// TIA Portal V19 program export: 1 tag tables, 0 data types, 17 data blocks, 13 code blocks (in call order from the OBs), 101 instance data blocks

VAR_GLOBAL   // PLC tag table "Default tag table"
   EMG_STOP AT %I0.0 : Bool;
   HOOTER_RESET AT %I0.1 : Bool;
   POWER_FAIL AT %I0.2 : Bool;
   "AIR PRESSURE FAIL" AT %I0.3 : Bool;
   "CENTRIFUGAL_PUMP-1_TRIP_(FWD)" AT %I0.4 : Bool;
   "CENTRIFUGAL_PUMP-2_TRIP_(RET)" AT %I0.5 : Bool;
   "FLOW SWITCH-1" AT %I0.6 : Bool;
   "FLOW SWITCH-2" AT %I0.7 : Bool;
   "LEVEL_SWITCH-1" AT %I1.0 : Bool;
   "LEVEL_SWITCH-2" AT %I1.1 : Bool;
   "LEVEL_SWITCH-3" AT %I1.2 : Bool;
   "LEVEL_SWITCH-4" AT %I1.3 : Bool;
   SPARE_DI1 AT %I1.4 : Bool;
   SPARE_DI2 AT %I1.5 : Bool;
   "CENTRIFUGAL_PUMP-1(FWD)" AT %Q0.0 : Bool;
   "CENTRIFUGAL_PUMP-2(RET)" AT %Q0.1 : Bool;
   "DOSING_PUMP-1" AT %Q0.2 : Bool;
   SPARE_DO1 AT %Q0.3 : Bool;
   HOOTER AT %Q0.4 : Bool;
   "PBV-125 PURIFIED WATER VESSEL OUTLET VALVE" AT %Q0.5 : Bool;
   "PBV-126 SOFT WATER VESSEL OUTLET VALVE" AT %Q0.6 : Bool;
   "PBV-127 PW INLET LINE" AT %Q0.7 : Bool;
   "PBV-128 PURIFIED WATER VESSEL–SPRAY BALL INLET LINE" AT %Q1.0 : Bool;
   "PBV-129 SOFT WATER VESSEL INLET LINE" AT %Q1.1 : Bool;
   "LEVEL_SWITCH-10" AT %I8.0 : Bool;
   AIR_PRESSURE_SWITCH AT %I8.1 : Bool;
   "PNEUMATIC_VALVE-7" AT %Q8.0 : Bool;
   "PNEUMATIC_VALVE-8" AT %Q8.1 : Bool;
   "PNEUMATIC_VALVE-9" AT %Q8.2 : Bool;
   "PNEUMATIC_VALVE-10" AT %Q8.3 : Bool;
   "PNEUMATIC_VALVE-11" AT %Q8.4 : Bool;
   "PNEUMATIC_VALVE-12" AT %Q8.5 : Bool;
   "PNEUMATIC_VALVE-13" AT %Q8.6 : Bool;
   "PNEUMATIC_VALVE-14" AT %Q8.7 : Bool;
   "PNEUMATIC_VALVE-15" AT %Q12.0 : Bool;
   "PNEUMATIC_VALVE-16" AT %Q12.1 : Bool;
   "PNEUMATIC_VALVE-17" AT %Q12.2 : Bool;
   "PNEUMATIC_VALVE-18" AT %Q12.3 : Bool;
   "PNEUMATIC_VALVE-19" AT %Q12.4 : Bool;
   CT_SENSOR AT %IW128 : Int;
   TS_SENSOR_1 AT %IW130 : Int;
   TS_SENSOR_2 AT %IW132 : Int;
   "CENTRIFUGAL_PUMP-1_RPM" AT %QW128 : Int;
   "DOSING_PUMP-1(4-20mA)" AT %QW130 : Int;
   System_Byte AT %MB1 : Byte;
   FirstScan AT %M1.0 : Bool;
   DiagStatusUpdate AT %M1.1 : Bool;
   AlwaysTRUE AT %M1.2 : Bool;
   AlwaysFALSE AT %M1.3 : Bool;
   "PNEUMATIC_VALVE-20" AT %Q12.5 : Bool;
   "PNEUMATIC_VALVE-21" AT %Q12.6 : Bool;
   "PNEUMATIC_VALVE-22" AT %Q12.7 : Bool;
   "PZDV-1" AT %Q13.0 : Bool;
   "PZDV-2" AT %Q13.1 : Bool;
   "CIP IN" AT %Q13.2 : Bool;
   "CIP OUT" AT %Q13.3 : Bool;
   "PH NOT ACHIEVED POPUP" AT %M100.0 : Bool;
   "PH ACHIEVED POPUP" AT %M100.1 : Bool;
   ALARM_1 AT %M20.0 : Bool;
   P_TRIG AT %M300.0 : Bool;
   ALARM_2 AT %M20.1 : Bool;
   ALARM_3 AT %M20.2 : Bool;
   ALARM_4 AT %M20.3 : Bool;
   ALARM_5 AT %M20.4 : Bool;
   P_TRIG_1 AT %M300.1 : Bool;
   P_TRIG_2 AT %M300.2 : Bool;
   P_TRIG_3 AT %M300.3 : Bool;
   P_TRIG_4 AT %M300.4 : Bool;
   P_TRIG_5 AT %M300.5 : Bool;
   ALARM_6 AT %M20.5 : Bool;
   ALARM_7 AT %M20.6 : Bool;
   P_TRIG_6 AT %M300.6 : Bool;
   P_TRIG_7 AT %M300.7 : Bool;
   ALARM_8 AT %M20.7 : Bool;
   P_TRIG_8 AT %M301.0 : Bool;
   P_TRIG_9 AT %M301.1 : Bool;
   "RINSE-1_START_POPUP" AT %M2.0 : Bool;
   "RINSE-1 RECIRCULATION_OR_DRAIN" AT %M2.1 : Bool;
   PH_ACHIEVED AT %M2.3 : Bool;
   "RINSE-2_START_POPUP" AT %M2.5 : Bool;
   PH_NOT_ACHIEVED AT %M2.4 : Bool;
   POPUPS AT %MW2 : Word;
   "FRESH CYCLE BIT" AT %M70.0 : Bool;
   "HEATING TEMPERATURE" AT %MD4 : Real;
   "HYSTERSIS ANS" AT %MD8 : Real;
   "HEATING BIT ON" AT %M70.1 : Bool;
   Tag_1 AT %QW96 : Int;
   "PUPM-1_SPEED" AT %MD12 : Real;
   ALARM AT %MW200 : Word;
   "ALAKLI / ACID_START" AT %M2.2 : Bool;
   "RINSE-2_RECIRCULATE_OR_DRAIN" AT %M2.6 : Bool;
   "RINSE-3_RECIRCULATION_OR_DRAIN" AT %M3.0 : Bool;
   FINAL_RINSE_START AT %M3.1 : Bool;
   CONDUCTIVITY_ACHIEVED AT %M3.2 : Bool;
   CONDUCTIVITY_NOT_ACHIEVED_RECIRCULATION_OR_FRESH_CYCLE AT %M3.3 : Bool;
   GOING_TO_FRESH_CYCLE AT %M3.4 : Bool;
   ALARM_9 AT %M21.0 : Bool;
   ERROR AT %M80.0 : Bool;
   "REST TESTYT" AT %M11.0 : Bool;
   PTRIG_10 AT %M11.1 : Bool;
   "RINSE-3_START" AT %M2.7 : Bool;
   ALKALI_LOW_LEVEL_POPUP AT %M3.5 : Bool;
   ACID_LOW_LEVEL_POPUP AT %M3.6 : Bool;
   RESET AT %M0.0 : Bool;
   ALKALI_BIT AT %M0.1 : Bool;
   ACID_BIT AT %M0.2 : Bool;
   "ALAKLI / ACID FRESH CYCLE" AT %M0.3 : Bool;
   "ALKALI/ ACID SELECT_POPUP" AT %M3.7 : Bool;
   "ALKALI / ACID DRAIN_SET" AT %M0.4 : Bool;
   FINAL_RINSE_DRAIN_SET AT %M0.5 : Bool;
   CONDUCTIVITY_ACHIEVED_BIT AT %M0.6 : Bool;
   CONDUCTIVITY_NOT_ACHIEVED_BIT AT %M0.7 : Bool;
   ALARM_10 AT %M21.1 : Bool;
   CYCLE_PAUSE_LSW_FWD AT %M16.0 : Bool;
   CYCLE_PAUSE_LSW_RET AT %M16.1 : Bool;
   AUTO_RESET AT %M16.2 : Bool;
   "RINSE-1_OVER" AT %M17.0 : Bool;
   "ALKALI / ACID_OVER" AT %M17.1 : Bool;
   "RINSE-2_OVER" AT %M17.2 : Bool;
   "FINAL RINSE-1_OVER" AT %M17.3 : Bool;
   "FINAL RINSE-2_OVER" AT %M17.4 : Bool;
   PTRIG_11 AT %M16.3 : Bool;
   PTRIG_12 AT %M16.4 : Bool;
   PTRIG_13 AT %M16.5 : Bool;
   PTRIG_14 AT %M16.6 : Bool;
   PTRIG_15 AT %M16.7 : Bool;
   CYCLE_OVER_ALARM AT %MW17 : Word;
   "CYCLE PAUSE" AT %M19.0 : Bool;
   VACCUME_VALVE_AUTO_BIT AT %M19.1 : Bool;
   N_TRIG AT %M19.2 : Bool;
   P_TRIG_10 AT %M301.2 : Bool;
   ALARM_11 AT %M21.2 : Bool;
   ALARM_12 AT %M21.3 : Bool;
   P_TRIG_11 AT %M301.3 : Bool;
   PTRIG_16 AT %M19.3 : Bool;
   PTRIG_17 AT %M19.4 : Bool;
   N_TRIG1 AT %M19.5 : Bool;
   N_TRIG2 AT %M19.6 : Bool;
   "TRIGGER 1" AT %M19.7 : Bool;
   "SET PRINT BIT" AT %M21.4 : Bool;
   "TAG SET" AT %M21.5 : Bool;
   LENGTH AT %MW22 : Int;
   TRIGGER AT %M70.3 : Bool;
   "EMG TRIG" AT %M24.0 : Bool;
   "AL1 REQ" AT %M24.1 : Bool;
   "AL2 REQ" AT %M24.2 : Bool;
   POWER_TRIG AT %M24.3 : Bool;
   "AL3 REQ" AT %M24.4 : Bool;
   "FWD TRIP_TRIG" AT %M24.5 : Bool;
   "AL4 REQ" AT %M24.6 : Bool;
   "RET TRIP_TRIG" AT %M24.7 : Bool;
   "AL5 REQ" AT %M25.0 : Bool;
   ALKALI_LL_TRIG AT %M25.1 : Bool;
   "AL6 REQ" AT %M25.2 : Bool;
   ACID_LL_TRIG AT %M25.3 : Bool;
   "AL7 REQ" AT %M25.4 : Bool;
   PWT_LL_TRIG AT %M25.5 : Bool;
   "AL8 REQ" AT %M25.6 : Bool;
   SWT_LL_TRIG AT %M25.7 : Bool;
   "AL9 REQ" AT %M26.0 : Bool;
   AIR_TRIG AT %M26.1 : Bool;
   FLS_TRIG AT %M26.2 : Bool;
   "AL10 REQ" AT %M26.3 : Bool;
   "AL11 REQ" AT %M26.4 : Bool;
   RLS_TRIG AT %M26.5 : Bool;
   PRODUCT_NAME AT %IB0 : Char;
   "PROD LENGTH" AT %MW28 : Int;
   "ADD PROD LENGTH" AT %MW30 : Int;
   "EQP LENGTH" AT %MW32 : Int;
   "ADD EQP LENGTH" AT %MW34 : Int;
   "OP LENGTH" AT %MW36 : Int;
   "ADD OP LENGTH" AT %MW38 : Int;
   "BATCH LENGTH" AT %MW40 : Int;
   "BATCH ACTUAL LENGTH" AT %MW42 : Int;
   "RECIPE LENGTH" AT %MW44 : Int;
   "ADD RECIPE LENGTH" AT %MW46 : Int;
   "EMP LENGTH" AT %MW48 : Int;
   "ADD EMP LENGTH" AT %MW50 : Int;
   N_TRIG3 AT %M21.6 : Bool;
   FOOTER AT %M21.7 : Bool;
   P_TRIG20 AT %M26.6 : Bool;
   PNV25 AT %Q13.4 : Bool;
   "SW TANK_START_POPUP" AT %M27.0 : Bool;
   "PW TANK_START_POPUP" AT %M27.1 : Bool;
   "SW TANK_OVER" AT %M27.2 : Bool;
   "PW TANK_OVER" AT %M27.3 : Bool;
   P_TRIG_12 AT %M26.7 : Bool;
   P_TRIG_13 AT %M27.4 : Bool;
   xyz AT %M27.5 : Bool;
   ON AT %M27.6 : Bool;
   ON1 AT %M27.7 : Bool;
   on2 AT %M52.0 : Bool;
   on4 AT %M52.1 : Bool;
   "PASSWORD DB" AT %MW54 : Int;
   "ACK 6MONTH" AT %M52.2 : Bool;
   "ACK 8MONTH" AT %M52.3 : Bool;
   "POPUP FOR 6 MONTH" AT %M52.4 : Bool;
   "POPUP FOR 8 MONTH" AT %M52.5 : Bool;
   "POPUP BIT TRIG" AT %M52.6 : Bool;
   "PBV-130 SOFT WATER VESSEL–SPRAY BALL INLET LINE" AT %Q14.0 : Bool;
   "PBV-131 DOSING PUMP INLET LINE" AT %Q14.1 : Bool;
   "PBV-132 PURIFIED WATER VESSEL OUTLET LINE" AT %Q14.2 : Bool;
   "PBV-133 SOFT WATER VESSEL OUTLET LINE" AT %Q14.3 : Bool;
   "PBV-134 FORWARD PUMP INLET LINE" AT %Q14.4 : Bool;
   "PBV-135 REVERSE PUMP CASING DRAIN" AT %Q14.5 : Bool;
   "PBV-136 FORWARD PUMP RECIRCULATION LINE" AT %Q14.6 : Bool;
   "PBV-137 FORWARD PUMP TO HEAT EXCHANGER LINE" AT %Q14.7 : Bool;
   "PBV-138 PURIFIED WATER DRAIN LINE" AT %Q15.0 : Bool;
   "PAV-139 HEAT EXCHANGER BYPASS DRAIN" AT %Q15.1 : Bool;
   "PBV-140 HEAT EXCHANGER INLET LINE" AT %Q15.2 : Bool;
   "PAV-141 STEAM INLET LINE" AT %Q15.3 : Bool;
   "PBV-142 FORWARD PUMP RECIRCULATION LINE" AT %Q15.4 : Bool;
   "PBV-143 FORWARD PUMP TO VESSEL INLET LINE" AT %Q15.5 : Bool;
   "PBV-144 VESSEL INLET LINE" AT %Q16.0 : Bool;
   "PBV-145 REVERSE PUMP TO VESSEL RECIRCULATION LINE" AT %Q16.1 : Bool;
   "PBV-146 REVERSE PUMP TO DRAIN LINE" AT %Q16.2 : Bool;
   "PBV-147 REVERSE PUMP CASING DRAIN LINE" AT %Q16.3 : Bool;
   "PBV-148 REVERSE PUMP INLET LINE" AT %Q16.4 : Bool;
   "PBV-157 SOFT WATER DRAIN LINE" AT %Q16.5 : Bool;
   "PBV-158 SOFT WATER VENT VALVE" AT %Q16.6 : Bool;
   "PBV-159 PURIFIED VENT VALVE" AT %Q16.7 : Bool;
   "PBV-160 ALKALI VALVE" AT %Q17.0 : Bool;
   "PBV-161 ACID VALVE" AT %Q17.1 : Bool;
   SPARE_DO4 AT %Q17.2 : Bool;
   SPARE_DO5 AT %Q17.3 : Bool;
   SPARE_DO6 AT %Q17.4 : Bool;
   SPARE_DO7 AT %Q17.5 : Bool;
   SPARE_DO8 AT %Q17.6 : Bool;
   SPARE_DO9 AT %Q17.7 : Bool;
   SPARE_DO2 AT %Q15.6 : Bool;
   SPARE_DO3 AT %Q15.7 : Bool;
   PH_SENSOR AT %IW134 : Int;
END_VAR

DATA_BLOCK "BATCH DATA"   // DB171
{ S7_Optimized_Access := 'FALSE' }
   VAR
      PRODUCT_NAME : String[30] := '  PRODUCT NAME             :  ';
      PRODUCT_NAME_CONCATE : String[80];
      BATCH_NO : String[30] := '  BATCH NO                 :  ';
      BATCH_NO_CONCATE : String[80];
      EQUIPMENT_ID_NO : String[30] := '  EQUIPMENT ID NO          :  ';
      EQUIPMENT_ID_NO_CONCATE : String[80];
      RECIPE_NO : String[30] := '  RECIPE NO                :  ';
      RECIPE_NO_CONCATE : String[80];
      OPERATOR_NAME : String[30] := '  OPERATOR NAME            :  ';
      OPERATOR_NAME_CONCATE : String[80];
      EMPLOYE_CODE : String[30] := '  EMPLOYE CODE             :  ';
      EMPLOYE_CODE_CONCATE : String[80];
   END_VAR
BEGIN
END_DATA_BLOCK

DATA_BLOCK "BUFFER"   // DB26
{ S7_Optimized_Access := 'FALSE' }
   VAR
      HMI_START : Bool;
      HMI_STOP : Bool;
      "MODE SELECTION" : Int;
      PROCESS : Int;
      Static_1 : Int;
      HMI_AUTO : Bool;
      HMI_MANUAL : Bool;
      HMI_STANDBY : Bool;
      "RECIPE DOWNLOAD" : Bool;
      "LEVEL BUFFER SWT" : Int;
      "LEVEL BUFFER PWT" : Int;
      "RINSE-1" : Int;
      "ACID / ALAKLI" : Int;
      "RINSE-2" : Int;
      "RINSE-3" : Int;
      FINAL_RINSE : Int;
      CONTINUE : Bool;
      RESET : Bool;
      phMAINTAIN : Bool;
   END_VAR
BEGIN
END_DATA_BLOCK

DATA_BLOCK "CYCLE_POPUP"   // DB37
{ S7_Optimized_Access := 'FALSE' }
   VAR
      "RINSE-1_START_YES" : Bool;
      "RINSE-1_START_NO" : Bool;
      "RINSE-1_RECIRCULATION" : Bool;
      "RINSE-1_DRAIN" : Bool;
      "RINSE-2_START_YES" : Bool;
      "RINSE-2_START_NO" : Bool;
      "RINSE-2_RECIRCULATION" : Bool;
      "RINSE-2_DRAIN" : Bool;
      "ACID/ALKALI_START_YES" : Bool;
      "ACID/ALKALI_START_NO" : Bool;
      "ALKALI/ACID_RECIRCULATION" : Bool;
      "ALKALI/ACID_DRAIN" : Bool;
      "ACID/ALKALI CONTINUE CYCLE" : Bool;
      "RINSE-3_START_YES" : Bool;
      "RINSE-3_START_NO" : Bool;
      "RINSE-3_RECIRCULATION" : Bool;
      "RINSE-3_DRAIN" : Bool;
      FINAL_RINSE_START_YES : Bool;
      FINAL_RINSE_START_NO : Bool;
      FINAL_RINSE_RECIRCULATION : Bool;
      FINAL_RINSE_FRESH_CYCLE : Bool;
      ALKALI : Bool;
      ACID : Bool;
      "ALKALI /ACID FRESH CYCLE" : Bool;
      FINAL_RINSE_DRAIN : Bool;
      "SW TANK_START_YES" : Bool;
      "SW TANK_START_NO" : Bool;
      "PW TANK_START_YES" : Bool;
      "PW TANK_START_NO" : Bool;
      "PW TANK_START_YES1" : Bool;
   END_VAR
BEGIN
END_DATA_BLOCK

DATA_BLOCK "DATE& TIME_DB"   // DB10
{ S7_Optimized_Access := 'TRUE' }
// stored: MemoryReserve 100
   VAR RETAIN
      READ : DTL;
      WRITE : DTL;
   END_VAR
   VAR
      SET : Bool;
      READ_DATE : Int;
      WRITE__DATE : Int;
   END_VAR
BEGIN
END_DATA_BLOCK

DATA_BLOCK "DATE_AND_TIME"   // DB5
{ S7_Optimized_Access := 'FALSE' }
   VAR
      SET_YEAR : DWord;
      SET_MONTH : DWord;
      SET_DAY : DWord;
      SET_HOUR : DWord;
      SET_MIN : DWord;
      SET_SEC : DWord;
   END_VAR
BEGIN
END_DATA_BLOCK

DATA_BLOCK "HEADER_DATA"   // DB170
{ S7_Optimized_Access := 'TRUE' }
// stored: MemoryReserve 100
BEGIN
END_DATA_BLOCK

DATA_BLOCK "HMI"   // DB86
{ S7_Optimized_Access := 'TRUE' }
// stored: MemoryReserve 100
   VAR
      HOOTER_RESET : Bool;
      M1_SUGAR : Bool;
      M1_MFG : Bool;
      M1_STORAGE_1 : Bool;
      M1_STORAGE_2 : Bool;
      M1_MIXING : Bool;
      M2_MFG : Bool;
      M2_STORAGE_1 : Bool;
      M2_STORAGE_2 : Bool;
      M2_MIXING : Bool;
   END_VAR
BEGIN
END_DATA_BLOCK

DATA_BLOCK "IN"   // DB28
{ S7_Optimized_Access := 'FALSE' }
   VAR
      EMG_STOP : Bool;
      HOOTER_RESET : Bool;
      POWER_FAIL : Bool;
      "PUMP-1_TRIP" : Bool;
      "PUMP-2_TRIP" : Bool;
      SWT_LL : Bool;
      SWT_ML : Bool;
      SWT_HL : Bool;
      PWT_LL : Bool;
      PWT_ML : Bool;
      PWT_HL : Bool;
      ALKALI_LL : Bool;
      ALAKLI_HL : Bool;
      ACID_LL : Bool;
      ACID_HL : Bool;
      LSW_FWD_PUMP : Bool;
      LSW_RET_PUMP : Bool;
      AIR_SWITCH : Bool;
      CT_SENSOR : Int;
      PH_SENSOR : Int;
      TEMP_SENSOR : Int;
   END_VAR
BEGIN
END_DATA_BLOCK

DATA_BLOCK "MANUAL BIT"   // DB1
{ S7_Optimized_Access := 'FALSE' }
   VAR
      HOOTER : Bool;
      "PUMP-1" : Bool;
      "PUMP-2" : Bool;
      DS_PUMP : Bool;
      "PNV-1" : Bool;
      "PNV-2" : Bool;
      "PNV-3" : Bool;
      "PNV-4" : Bool;
      "PNV-5" : Bool;
      "PNV-6" : Bool;
      "PNV-7" : Bool;
      "PNV-8" : Bool;
      "PNV-9" : Bool;
      "PNV-10" : Bool;
      "PNV-11" : Bool;
      "PNV-12" : Bool;
      "PNV-13" : Bool;
      "PNV-14" : Bool;
      "PNV-15" : Bool;
      "PNV-16" : Bool;
      "PNV-17" : Bool;
      "PNV-18" : Bool;
      "PNV-19" : Bool;
      "PNV-20" : Bool;
      "PNV-21" : Bool;
      "PNV-22" : Bool;
      "PZDV-1" : Bool;
      "PZDV-2" : Bool;
      CIP_IN : Bool;
      CIP_OUT : Bool;
      "PNV-25" : Bool;
   END_VAR
BEGIN
END_DATA_BLOCK

DATA_BLOCK "MODE SELECTION"   // DB27
{ S7_Optimized_Access := 'FALSE' }
   VAR
      AUTO : Bool;
      MANUAL : Bool;
      STANDBY : Bool;
      "MODE BUFFER" : Int;
   END_VAR
BEGIN
END_DATA_BLOCK

DATA_BLOCK "OP"   // DB29
{ S7_Optimized_Access := 'FALSE' }
   VAR
      HOOTER : Bool;
      "PUMP-1" : Bool;
      "PUMP-2" : Bool;
      DS_PUMP : Bool;
      "PNV-1" : Bool;
      "PNV-2" : Bool;
      "PNV-3" : Bool;
      "PNV-4" : Bool;
      "PNV-5" : Bool;
      "PNV-6" : Bool;
      "PNV-7" : Bool;
      "PNV-8" : Bool;
      "PNV-9" : Bool;
      "PNV-10" : Bool;
      "PNV-11" : Bool;
      "PNV-12" : Bool;
      "PNV-13" : Bool;
      "PNV-14" : Bool;
      "PNV-15" : Bool;
      "PNV-16" : Bool;
      "PNV-17" : Bool;
      "PNV-18" : Bool;
      "PNV-19" : Bool;
      "PNV-20" : Bool;
      "PNV-21" : Bool;
      "PNV-22" : Bool;
      "PZDV-1" : Bool;
      "PZDV-2" : Bool;
      CIP_IN : Bool;
      CIP_OUT : Bool;
      "PNV-25" : Bool;
   END_VAR
BEGIN
END_DATA_BLOCK

DATA_BLOCK "PRINT"   // DB134
{ S7_Optimized_Access := 'TRUE' }
// stored: MemoryReserve 100
   VAR RETAIN
      "PRINT START" : Bool;
   END_VAR
   VAR
      "PRESENT VALUE" : Int;
   END_VAR
   VAR RETAIN
      INTERVAL : Int;
   END_VAR
BEGIN
END_DATA_BLOCK

DATA_BLOCK "PRINTING DATA"   // DB133
{ S7_Optimized_Access := 'FALSE' }
   VAR
      "LINE 1" : String[80] := '                          M/S PHARMAFORCE LAB UNIT-II                       ';
      "LINE 2" : String[80] := '                 MFG BY : KOTHARI PHARMA TECHNOLOGIES  PVT LTD              ';
      "LINE 3" : String[80] := ' -------------------------------------------------------------------------------';
      "LINE 4" : String[80] := '                                     CIP SKID                                 ';
      "LINE 5" : String[80] := ' -------------------------------------------------------------------------------';
      "LINE 6" : String[80] := '    /  /              RINSE-1,RINSE-2, FINAL RINSE-1 PARAMETER    ';
      "LINE 7" : String[80] := ' -------------------------------------------------------------------------------';
      "LINE 8" : String[80] := '  PARAMETER                        SET VALUE';
      "LINE 9" : String[80] := '                                   RINSE-1          RINSE-2          F_RINSE-1';
      "LINE 10" : String[80] := '  HEATING TEMPERATURE  ';
      "LINE 11" : String[80] := '  CLEANING TIME ';
      "LINE 12" : String[80] := '  RECIRCULATION TIME ';
      "LINE 13" : String[80] := '  DRAIN TIME';
      "LINE 14" : String[80] := '  PUMP CASING DRAIN TIME ';
      "LINE 15" : String[80] := '  FWD PUMP HEATING RPM ';
      "LINE 16" : String[80] := '  FWD PUMP CLEANING RPM ';
      "LINE 17" : String[80];
      "LINE 18" : String[80] := ' -------------------------------------------------------------------------------';
      "LINE 19" : String[80] := '    /  /              ALKALI / ACID PARAMETER ';
      "LINE 20" : String[80] := ' -------------------------------------------------------------------------------';
      "LINE 21" : String[80] := '  PARAMETER                             SET VALUE                 ';
      "LINE 22" : String[80] := '  HEATING TEMPERATURE  ';
      "LINE 23" : String[80] := '  CLEANING TIME ';
      "LINE 24" : String[80] := '  RECIRCULATION TIME ';
      "LINE 25" : String[80] := '  DRAIN TIME';
      "LINE 26" : String[80] := '  PUMP CASING DRAIN TIME ';
      "LINE 27" : String[80] := '  FWD PUMP HEATING RPM ';
      "LINE 28" : String[80] := '  FWD PUMP CLEANING RPM ';
      "LINE 29" : String[80] := '  BEFORE CLEANING PH LOW ';
      "LINE 30" : String[80] := '  BEFORE CLEANING PH HIGH ';
      "LINE 31" : String[80] := '  AFTER CLEANING PH LOW ';
      "LINE 32" : String[80] := '  AFTER CLEANING PH HIGH ';
      "LINE 33" : String[80];
      "LINE 34" : String[80] := ' -------------------------------------------------------------------------------';
      "LINE 35" : String[80] := '    /  /              FINAL RINSE-2 PARAMETER    ';
      "LINE 36" : String[80] := ' -------------------------------------------------------------------------------';
      "LINE 37" : String[80] := '  PARAMETER                            SET VALUE                   ';
      "LINE 38" : String[80] := '  HEATING TEMPERATURE  ';
      "LINE 39" : String[80] := '  CLEANING TIME ';
      "LINE 40" : String[80] := '  RECIRCULATION TIME ';
      "LINE 41" : String[80] := '  DRAIN TIME';
      "LINE 42" : String[80] := '  PUMP CASING DRAIN TIME ';
      "LINE 43" : String[80] := '  FWD PUMP HEATING RPM ';
      "LINE 44" : String[80] := '  FWD PUMP CLEANING RPM ';
      "LINE 45" : String[80] := '  CONDUCTIVITY ';
      "LINE 46" : String[80];
      "LINE 47" : String[80];
      AL1 : String[80] := '      :  :        EMERGENCY PRESSED ';
      AL2 : String[80] := '      :  :        POWER FAIL ';
      AL3 : String[80] := '      :  :        FORWARD PUMP TRIP';
      AL4 : String[80] := '      :  :        RETURN PUMP TRIP';
      AL5 : String[80] := '      :  :        ALKALI LEVEL IS LOW';
      AL6 : String[80] := '      :  :        ACID LEVEL IS LOW';
      AL7 : String[80] := '      :  :        PURE WATER LEVLE IS LOW ';
      AL8 : String[80] := '      :  :        SOFTWATER LEVLE IS LOW ';
      AL9 : String[80] := '      :  :        AIR FAIL';
      AL10 : String[80] := '      :  :        FORWARD LIMIT SWITCH IS UNHEALTHY';
      AL11 : String[80] := '      :  :        RETURN LIMIT SWITCH IS UNHEALTHY';
      AL12 : String[80];
      PV1 : String[80] := ' -------------------------------------------------------------------------------';
      PV2 : String[80] := '    /  /              PRESENT VALUES    ';
      PV3 : String[80] := ' -------------------------------------------------------------------------------';
      PV4 : String[80] := '                     TEMP           PUMP-1_RPM           PH          CON ';
      PV5 : String[80] := '      :  :        ';
      BLANK : String[80] := '.                                                            ';
      FOOTER1 : String[80] := '  DONE BY :                                  CHECKED BY :                  ';
   END_VAR
BEGIN
END_DATA_BLOCK

DATA_BLOCK "RECIPE DB"   // DB9
{ S7_Optimized_Access := 'FALSE' }
   VAR
      "RINSE-1_CLEANING_TIME_SV" : Int;
      "RINSE-1_RECIRCULATION_TIME_SV" : Int;
      "RINSE-1_DRAIN_TIME_SV" : Int;
      "RINSE-1_PUMP_CHASING_TIME_SV" : Int;
      "RINSE-1_TEMPERATURE_SET" : Real;
      "RINSE-1_FWD_PUMP_HEATING_RPM" : Int;
      "RINSE-1_FWD_PUMP_CLEANING_RPM" : Int;
      "RINSE-2_TEMPERATURE_SET" : Real;
      "RINSE-2_CLEANING_TIME_SV" : Int;
      "RINSE-2_RECIRCULATION_TIME_SV" : Int;
      "RINSE-2_DRAIN_TIME_SV" : Int;
      "RINSE-2_PUMP_CHASING_TIME_SV" : Int;
      "RINSE-2_FWD_PUMP_HEATING_RPM" : Int;
      "RINSE-2_FWD_PUMP_CLEANING_RPM" : Int;
      DOSING_TIME_SV : Int;
      "ALKALI/ACID_TEMPERATURE_SET" : Real;
      "ALKALI/ACID_CLEANING_TIME_SV" : Int;
      "ALKALI/ACID_RECIRCULATION_TIME_SV" : Int;
      "ALKALI/ACID_DRAIN_TIME_SV" : Int;
      "ALKALI/ACID_PUMP_CHASING_TIME_SV" : Int;
      "ALKALI/ACID_FWD_PUMP_HEATING_RPM" : Int;
      "ALKALI/ACID_FWD_PUMP_CLEANING_RPM" : Int;
      FINAL_RINSE_TEMPERATURE_SET : Real;
      FINAL_RINSE_CLEANING_TIME_SV : Int;
      FINAL_RINSE_RECIRCULATION_TIME_SV : Int;
      FINAL_RINSE_DRAIN_TIME_SV : Int;
      FINAL_RINSE_PUMP_CHASING_TIME_SV : Int;
      "FINAL_RINSE-2_FWD_PUMP_HEATING_RPM" : Int;
      "FINAL_RINSE-2_FWD_PUMP_CLEANING_RPM" : Int;
      CONDUCTIVITY_SET : Real;
      "PH_SET (NOT USED)" : Int;
      DOSING_PH_LOW : Real;
      DOSING_PH_HIGH : Real;
      "RINSE-3_TEMPERATURE_SET" : Real;
      "RINSE-3_CLEANING_TIME_SV" : Int;
      "RINSE-3_RECIRCULATION_TIME_SV" : Int;
      "RINSE-3_DRAIN_TIME_SV" : Int;
      "RINSE-3_PUMP_CHASING_TIME_SV" : Int;
      "FINAL_RINSE-1_FWD_PUMP_HEATING_RPM" : Int;
      "FINAL_RINSE-1_FWD_PUMP_CLEANING_RPM" : Int;
      SET_TEMPERATURE : Real;
      "RINSE-1_SELECT" : Bool;
      "ALKALI / ACID_SELECT" : Bool;
      "RINSE-2_SELECT" : Bool;
      "FINAL_RINSE-1_SELECT" : Bool;
      "FINAL_RINSE-2_SELECT" : Bool;
      RECIRCULATION_PH_LOW : Real;
      RECIRCULATION_PH_HIGH : Real;
      "SW TANK_SELECT" : Bool;
      "PW TANK_SELECT" : Bool;
      "SW TANK_FWD_PUMP_CLEANING_RPM" : Int;
      "PW TANK_FWD_PUMP_CLEANING_RPM" : Int;
      "SW TANK_TEMPERATURE_SET" : Real;
      "PW TANK_TEMPERATURE_SET" : Real;
      "SW TANK_CLEANING_TIME_SV" : Int;
      "SW TANK_DRAIN_TIME_SV" : Int;
      "SW TANK_PUMP_CHASING_TIME_SV" : Int;
      "PW TANK_CLEANING_TIME_SV" : Int;
      "PW TANK_DRAIN_TIME_SV" : Int;
      "PW TANK_PUMP_CHASING_TIME_SV" : Int;
   END_VAR
BEGIN
END_DATA_BLOCK

DATA_BLOCK "SCALE_SET"   // DB36
{ S7_Optimized_Access := 'FALSE' }
   VAR RETAIN
      CT_SCALE_MIN : Real;
      CT_SCALE_MAX : Real;
      PH_SCALE_MIN : Real;
      PH_SCALE_MAX : Real;
      TS_SCALE_MIN : Real;
      TS_SCALE_MAX : Real;
      CT_NORM : Real;
      PH_NORM : Real;
      TS_NORM : Real;
      CT_PV : Real;
      PH_PV : Real;
      TS_PV : Real;
      FWD_PUMP_SPEED : Real;
      HYSTERSIS : Real;
      "PUMP-1_MIN_SPEED" : Int;
      "PUMP-1_MAX_SPEED" : Int;
   END_VAR
BEGIN
END_DATA_BLOCK

DATA_BLOCK "SET_PARAMETERS"   // DB24
{ S7_Optimized_Access := 'FALSE' }
   VAR RETAIN
      "RINSE-1_CLEANING_TIME_SV" : Int;
      "RINSE-1_CLEANING_TIME_PV" : Int;
      "RINSE-1_RECIRCULATION_TIME_SV" : Int;
      "RINSE-1_RECIRCULATION_TIME_PV" : Int;
      "RINSE-1_DRAIN_TIME_SV" : Int;
      "RINSE-1_DRAIN_TIME_PV" : Int;
      "RINSE-1_PUMP_CHASING_TIME_SV" : Int;
      "RINSE-1_PUMP_CHASING_TIME_PV" : Int;
      "RINSE-1_TEMPERATURE_SET" : Real;
      "RINSE-2_TEMPERATURE_SET" : Real;
      "RINSE-2_CLEANING_TIME_SV" : Int;
      "RINSE-2_CLEANING_TIME_PV" : Int;
      "RINSE-2_RECIRCULATION_TIME_SV" : Int;
      "RINSE-2_RECIRCULATION_TIME_PV" : Int;
      "RINSE-2_DRAIN_TIME_SV" : Int;
      "RINSE-2_DRAIN_TIME_PV" : Int;
      "RINSE-2_PUMP_CHASING_TIME_SV" : Int;
      "RINSE-2_PUMP_CHASING_TIME_PV" : Int;
      DOSING_TIME_SV : Int;
      DOSING_TIME_PV : Int;
      "ALKALI/ACID_TEMPERATURE_SET" : Real;
      "ALKALI/ACID_CLEANING_TIME_SV" : Int;
      "ALKALI/ACID_CLEANING_TIME_PV" : Int;
      "ALKALI/ACID_RECIRCULATION_TIME_SV" : Int;
      "ALKALI/ACID_RECIRCULATION_TIME_PV" : Int;
      "ALKALI/ACID_DRAIN_TIME_SV" : Int;
      "ALKALI/ACID_DRAIN_TIME_PV" : Int;
      "ALKALI/ACID_PUMP_CHASING_TIME_SV" : Int;
      "ALKALI/ACID_PUMP_CHASING_TIME_PV" : Int;
      FINAL_RINSE_TEMPERATURE_SET : Real;
      FINAL_RINSE_CLEANING_TIME_SV : Int;
      FINAL_RINSE_CLEANING_TIME_PV : Int;
      FINAL_RINSE_RECIRCULATION_TIME_SV : Int;
      FINAL_RINSE_RECIRCULATION_TIME_PV : Int;
      FINAL_RINSE_DRAIN_TIME_SV : Int;
      FINAL_RINSE_DRAIN_TIME_PV : Int;
      FINAL_RINSE_PUMP_CHASING_TIME_SV : Int;
      FINAL_RINSE_PUMP_CHASING_TIME_PV : Int;
      CONDUCTIVITY_SET : Real;
      PH_SET : Real;
      DOSING_PH_LOW : Real;
      DOSING_PH_HIGH : Real;
      "RINSE-3_TEMPERATURE_SET" : Real;
      "RINSE-3_CLEANING_TIME_SV" : Int;
      "RINSE-3_CLEANING_TIME_PV" : Int;
      "RINSE-3_RECIRCULATION_TIME_SV" : Int;
      "RINSE-3_RECIRCULATION_TIME_PV" : Int;
      "RINSE-3_DRAIN_TIME_SV" : Int;
      "RINSE-3_DRAIN_TIME_PV" : Int;
      "RINSE-3_PUMP_CHASING_TIME_SV" : Int;
      "RINSE-3_PUMP_CHASING_TIME_PV" : Int;
      SET_TEMPERATURE : Real;
      "RINSE-1_FWD_PUMP_HEATING_RPM" : Int;
      "RINSE-1_FWD_PUMP_CLEANING_RPM" : Int;
      "RINSE-2_FWD_PUMP_HEATING_RPM" : Int;
      "RINSE-2_FWD_PUMP_CLEANING_RPM" : Int;
      "ALKALI/ACID_FWD_PUMP_HEATING_RPM" : Int;
      "ALKALI/ACID_FWD_PUMP_CLEANING_RPM" : Int;
      "FINAL_RINSE-2_FWD_PUMP_HEATING_RPM" : Int;
      "FINAL_RINSE-2_FWD_PUMP_CLEANING_RPM" : Int;
      "FINAL_RINSE-1_FWD_PUMP_HEATING_RPM" : Int;
      "FINAL_RINSE-1_FWD_PUMP_CLEANING_RPM" : Int;
      "PUMP-1_SPEED" : Int;
      RECIRCULATION_PH_LOW : Real;
      RECIRCULATION_PH_HIGH : Real;
      PLANT1_TANK_SELECT : Byte;
      PLANT_SELECT : Byte;
      PLANT2_TANK_SELECT : Byte;
      PLANT3_TANK_SELECT : Byte;
      "SW TANK_CLEANING_TIME_SV" : Int;
      "SW TANK_CLEANING_TIME_PV" : Int;
      "SW TANK_DRAIN_TIME_SV" : Int;
      "SW TANK_DRAIN_TIME_PV" : Int;
      "SW TANK_PUMP_CHASING_TIME_SV" : Int;
      "SW TANK_PUMP_CHASING_TIME_PV" : Int;
      "PW TANK_CLEANING_TIME_SV" : Int;
      "PW TANK_CLEANING_TIME_PV" : Int;
      "PW TANK_DRAIN_TIME_SV" : Int;
      "PW TANK_DRAIN_TIME_PV" : Int;
      "PW TANK_PUMP_CHASING_TIME_SV" : Int;
      "PW TANK_PUMP_CHASING_TIME_PV" : Int;
      "SW TANK_FWD_PUMP_CLEANING_RPM" : Int;
      "PW TANK_FWD_PUMP_CLEANING_RPM" : Int;
      "SW TANK_TEMPERATURE_SET" : Real;
      "PW TANK_TEMPERATURE_SET" : Real;
      DOSING_PH_LOW1 : Real;
      DOSING_PH_HIGH1 : Real;
   END_VAR
BEGIN
END_DATA_BLOCK

DATA_BLOCK "STRING"   // DB169
{ S7_Optimized_Access := 'FALSE' }
   VAR
      PRODUCT_NAME : String[50];
      BATCH_NO : String[50];
      EQUIPMENT_ID_NO : String[50];
      RECIPE_NO : String[50];
      OPERATOR_NAME : String[50];
      EMPLOYE_CODE : String[50];
   END_VAR
BEGIN
END_DATA_BLOCK

ORGANIZATION_BLOCK "Main"   // OB1, LAD, ProgramCycle
TITLE = "Main Program Sweep (Cycle)"
{ S7_Optimized_Access := 'TRUE' }
// stored: SetENOAutomatically false
   VAR_INPUT
      Initial_Call : Bool;   // Initial call of this OB
      Remanence : Bool;   // =True, if remanent data are available
   END_VAR
   VAR_TEMP   // added for the SCL form of the ladder/FBD networks
      _w1 : Bool;
      _w2 : Bool;
      _w3 : Bool;
      _w4 : Bool;
      _w5 : Bool;
      _w6 : Bool;
      _w7 : Bool;
      _w8 : Bool;
   END_VAR
BEGIN

REGION Network 1: MAIN BLOCK CALLING
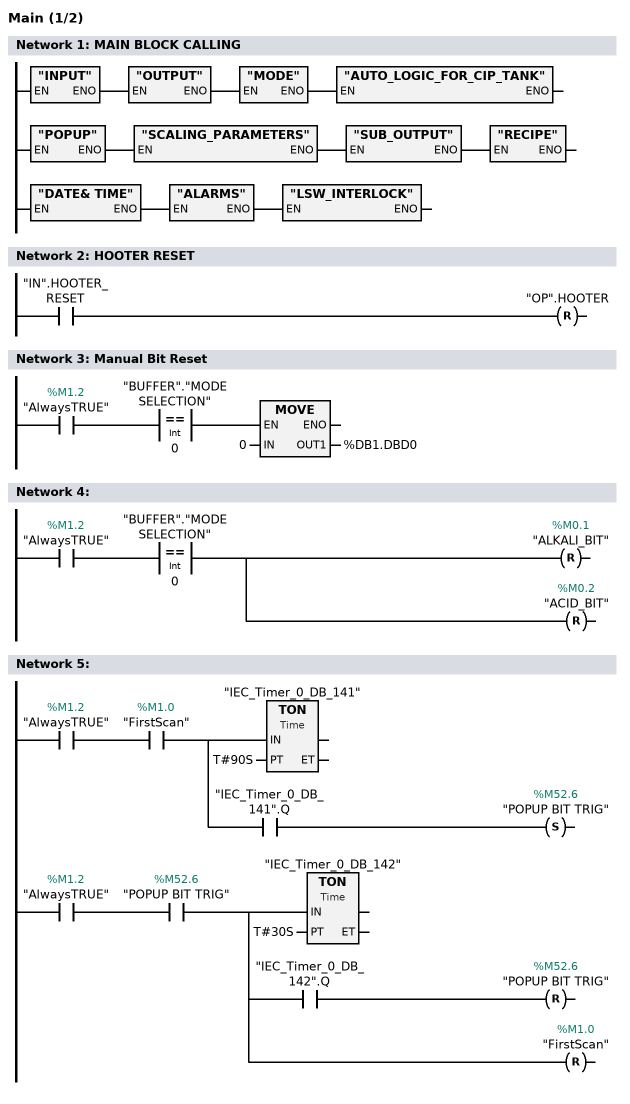
   RUNG wire#powerrail
      "INPUT"()
      "OUTPUT"()
      "MODE"()
      "AUTO_LOGIC_FOR_CIP_TANK"()
   END_RUNG
   RUNG wire#powerrail
      "POPUP"()
      "SCALING_PARAMETERS"()
      "SUB_OUTPUT"()
      "RECIPE"()
   END_RUNG
   RUNG wire#powerrail
      "DATE& TIME"()
      "ALARMS"()
      "LSW_INTERLOCK"()
   END_RUNG
   // the same network as SCL:
   "INPUT"(ENO => #_w1);
   "OUTPUT"(EN := #_w1, ENO => #_w2);
   "MODE"(EN := #_w2, ENO => #_w3);
   IF #_w3 THEN "AUTO_LOGIC_FOR_CIP_TANK"(); END_IF;
   "POPUP"(ENO => #_w4);
   "SCALING_PARAMETERS"(EN := #_w4, ENO => #_w5);
   "SUB_OUTPUT"(EN := #_w5, ENO => #_w6);
   IF #_w6 THEN "RECIPE"(); END_IF;
   "DATE& TIME"(ENO => #_w7);
   "ALARMS"(EN := #_w7, ENO => #_w8);
   IF #_w8 THEN "LSW_INTERLOCK"(); END_IF;
END_REGION

REGION Network 2: HOOTER RESET
   RUNG wire#powerrail
      Contact( "IN".HOOTER_RESET )
      R_Coil( "OP".HOOTER )
   END_RUNG
   // the same network as SCL:
   IF "IN".HOOTER_RESET THEN "OP".HOOTER := FALSE; END_IF;
END_REGION

REGION Network 3: Manual Bit Reset
   RUNG wire#powerrail
      Contact( "AlwaysTRUE" )
      { S7_Templates := "SrcType := Int" } EQ_Contact(in1 := "BUFFER"."MODE SELECTION", in2 := 0)
      Move(in := 0, out1 => %DB1.DBD0)
   END_RUNG
   // the same network as SCL:
   IF "AlwaysTRUE" AND ("BUFFER"."MODE SELECTION" = 0) THEN %DB1.DBD0 := 0; END_IF;
END_REGION

REGION Network 4
   RUNG wire#powerrail
      Contact( "AlwaysTRUE" )
      { S7_Templates := "SrcType := Int" } EQ_Contact(in1 := "BUFFER"."MODE SELECTION", in2 := 0)
      wire#w1
      R_Coil( "ALKALI_BIT" )
   END_RUNG
   RUNG wire#w1
      R_Coil( "ACID_BIT" )
   END_RUNG
   // the same network as SCL:
   IF "AlwaysTRUE" AND ("BUFFER"."MODE SELECTION" = 0) THEN
       "ALKALI_BIT" := FALSE;
       "ACID_BIT" := FALSE;
   END_IF;
END_REGION

REGION Network 5
   RUNG wire#powerrail
      Contact( "AlwaysTRUE" )
      Contact( "FirstScan" )
      wire#w1
      { S7_Templates := "time_type := Time" } "IEC_Timer_0_DB_141".TON(pt := T#90S, et =>)
   END_RUNG
   RUNG wire#w1
      Contact( "IEC_Timer_0_DB_141".Q )
      S_Coil( "POPUP BIT TRIG" )
   END_RUNG
   RUNG wire#powerrail
      Contact( "AlwaysTRUE" )
      Contact( "POPUP BIT TRIG" )
      wire#w2
      { S7_Templates := "time_type := Time" } "IEC_Timer_0_DB_142".TON(pt := T#30S, et =>)
   END_RUNG
   RUNG wire#w2
      Contact( "IEC_Timer_0_DB_142".Q )
      R_Coil( "POPUP BIT TRIG" )
   END_RUNG
   RUNG wire#w2
      R_Coil( "FirstScan" )
   END_RUNG
   // the same network as SCL:
   #_w1 := "AlwaysTRUE" AND "FirstScan";
   "IEC_Timer_0_DB_141".TON(IN := #_w1, PT := T#90S);
   IF #_w1 AND "IEC_Timer_0_DB_141".Q THEN "POPUP BIT TRIG" := TRUE; END_IF;
   #_w2 := "AlwaysTRUE" AND "POPUP BIT TRIG";
   "IEC_Timer_0_DB_142".TON(IN := #_w2, PT := T#30S);
   IF #_w2 AND "IEC_Timer_0_DB_142".Q THEN "POPUP BIT TRIG" := FALSE; END_IF;
   IF #_w2 THEN "FirstScan" := FALSE; END_IF;
END_REGION

REGION Network 6: 6 MONTH
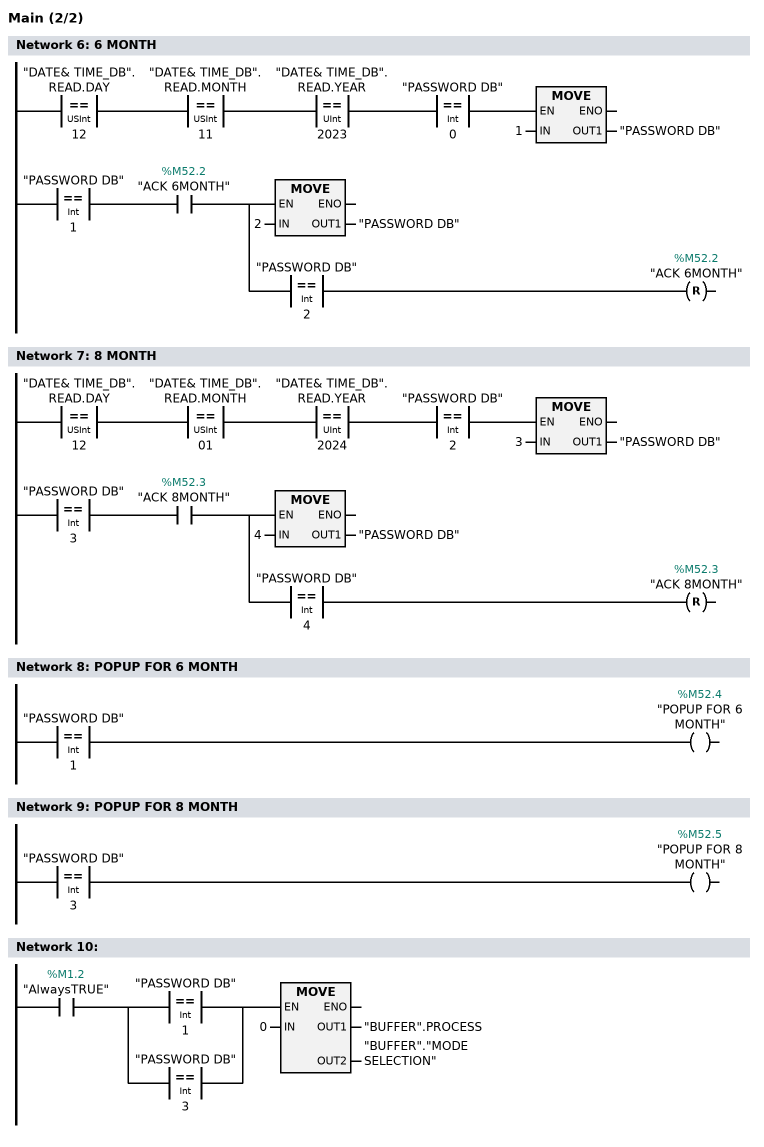
   RUNG wire#powerrail
      { S7_Templates := "SrcType := USInt" } EQ_Contact(in1 := "DATE& TIME_DB".READ.DAY, in2 := 12)
      { S7_Templates := "SrcType := USInt" } EQ_Contact(in1 := "DATE& TIME_DB".READ.MONTH, in2 := 11)
      { S7_Templates := "SrcType := UInt" } EQ_Contact(in1 := "DATE& TIME_DB".READ.YEAR, in2 := 2023)
      { S7_Templates := "SrcType := Int" } EQ_Contact(in1 := "PASSWORD DB", in2 := 0)
      Move(in := 1, out1 => "PASSWORD DB")
   END_RUNG
   RUNG wire#powerrail
      { S7_Templates := "SrcType := Int" } EQ_Contact(in1 := "PASSWORD DB", in2 := 1)
      Contact( "ACK 6MONTH" )
      wire#w1
      Move(in := 2, out1 => "PASSWORD DB")
   END_RUNG
   RUNG wire#w1
      { S7_Templates := "SrcType := Int" } EQ_Contact(in1 := "PASSWORD DB", in2 := 2)
      R_Coil( "ACK 6MONTH" )
   END_RUNG
   // the same network as SCL:
   IF ("DATE& TIME_DB".READ.DAY = 12) AND ("DATE& TIME_DB".READ.MONTH = 11) AND ("DATE& TIME_DB".READ.YEAR = 2023) AND ("PASSWORD DB" = 0) THEN
       "PASSWORD DB" := 1;
   END_IF;
   #_w1 := ("PASSWORD DB" = 1) AND "ACK 6MONTH";
   IF #_w1 THEN "PASSWORD DB" := 2; END_IF;
   IF #_w1 AND ("PASSWORD DB" = 2) THEN "ACK 6MONTH" := FALSE; END_IF;
END_REGION

REGION Network 7: 8 MONTH
   RUNG wire#powerrail
      { S7_Templates := "SrcType := USInt" } EQ_Contact(in1 := "DATE& TIME_DB".READ.DAY, in2 := 12)
      { S7_Templates := "SrcType := USInt" } EQ_Contact(in1 := "DATE& TIME_DB".READ.MONTH, in2 := 01)
      { S7_Templates := "SrcType := UInt" } EQ_Contact(in1 := "DATE& TIME_DB".READ.YEAR, in2 := 2024)
      { S7_Templates := "SrcType := Int" } EQ_Contact(in1 := "PASSWORD DB", in2 := 2)
      Move(in := 3, out1 => "PASSWORD DB")
   END_RUNG
   RUNG wire#powerrail
      { S7_Templates := "SrcType := Int" } EQ_Contact(in1 := "PASSWORD DB", in2 := 3)
      Contact( "ACK 8MONTH" )
      wire#w1
      Move(in := 4, out1 => "PASSWORD DB")
   END_RUNG
   RUNG wire#w1
      { S7_Templates := "SrcType := Int" } EQ_Contact(in1 := "PASSWORD DB", in2 := 4)
      R_Coil( "ACK 8MONTH" )
   END_RUNG
   // the same network as SCL:
   IF ("DATE& TIME_DB".READ.DAY = 12) AND ("DATE& TIME_DB".READ.MONTH = 01) AND ("DATE& TIME_DB".READ.YEAR = 2024) AND ("PASSWORD DB" = 2) THEN
       "PASSWORD DB" := 3;
   END_IF;
   #_w1 := ("PASSWORD DB" = 3) AND "ACK 8MONTH";
   IF #_w1 THEN "PASSWORD DB" := 4; END_IF;
   IF #_w1 AND ("PASSWORD DB" = 4) THEN "ACK 8MONTH" := FALSE; END_IF;
END_REGION

REGION Network 8: POPUP FOR 6 MONTH
   RUNG wire#powerrail
      { S7_Templates := "SrcType := Int" } EQ_Contact(in1 := "PASSWORD DB", in2 := 1)
      Coil( "POPUP FOR 6 MONTH" )
   END_RUNG
   // the same network as SCL:
   "POPUP FOR 6 MONTH" := "PASSWORD DB" = 1;
END_REGION

REGION Network 9: POPUP FOR 8 MONTH
   RUNG wire#powerrail
      { S7_Templates := "SrcType := Int" } EQ_Contact(in1 := "PASSWORD DB", in2 := 3)
      Coil( "POPUP FOR 8 MONTH" )
   END_RUNG
   // the same network as SCL:
   "POPUP FOR 8 MONTH" := "PASSWORD DB" = 3;
END_REGION

REGION Network 10
   RUNG wire#powerrail
      Contact( "AlwaysTRUE" )
      wire#w1
      { S7_Templates := "SrcType := Int" } EQ_Contact(in1 := "PASSWORD DB", in2 := 1)
      wire#w2
      Move(in := 0, out1 => "BUFFER".PROCESS, out2 => "BUFFER"."MODE SELECTION")
   END_RUNG
   RUNG wire#w1
      { S7_Templates := "SrcType := Int" } EQ_Contact(in1 := "PASSWORD DB", in2 := 3)
   END_RUNG wire#w2
   // the same network as SCL:
   IF "AlwaysTRUE" AND (("PASSWORD DB" = 1) OR ("PASSWORD DB" = 3)) THEN
       "BUFFER".PROCESS := 0;
       "BUFFER"."MODE SELECTION" := 0;
   END_IF;
END_REGION
END_ORGANIZATION_BLOCK

FUNCTION "INPUT" : Void   // FC2, LAD
{ S7_Optimized_Access := 'TRUE' }
// stored: SetENOAutomatically false
BEGIN

REGION Network 1: EMERGENCY_STOP
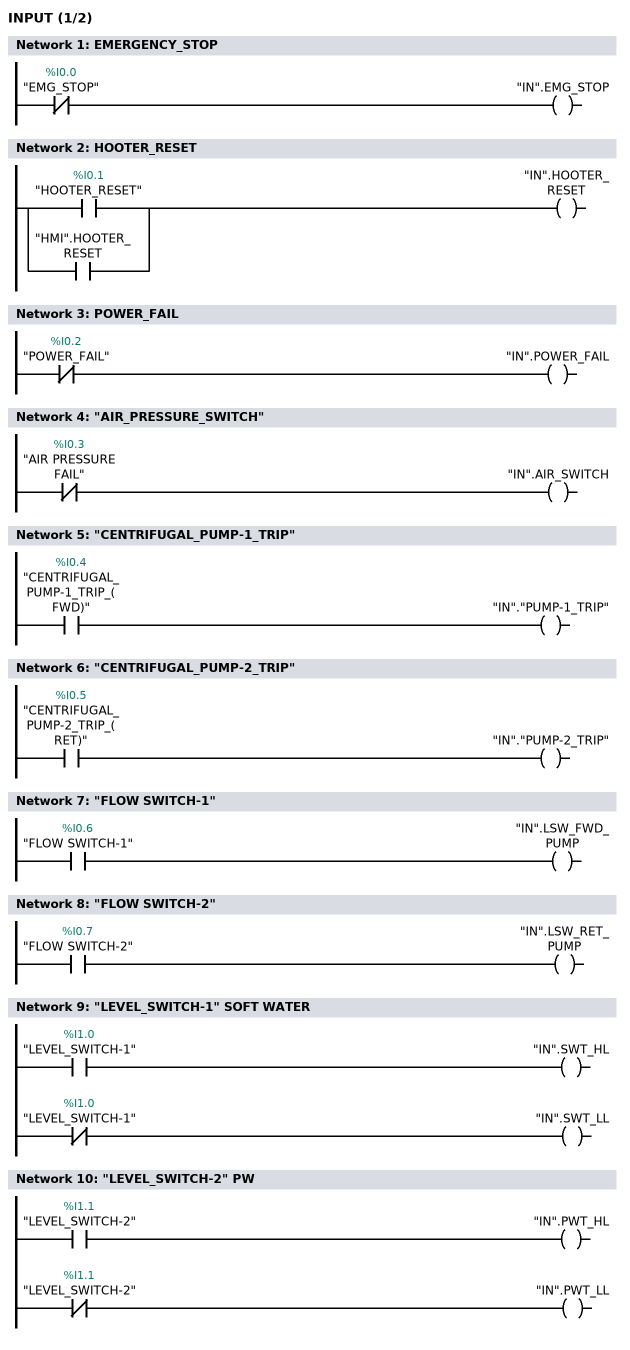
   RUNG wire#powerrail
      I_Contact( "EMG_STOP" )
      Coil( "IN".EMG_STOP )
   END_RUNG
   // the same network as SCL:
   "IN".EMG_STOP := NOT "EMG_STOP";
END_REGION

REGION Network 2: HOOTER_RESET
   RUNG wire#powerrail
      Contact( "HOOTER_RESET" )
      wire#w1
      Coil( "IN".HOOTER_RESET )
   END_RUNG
   RUNG wire#powerrail
      Contact( "HMI".HOOTER_RESET )
   END_RUNG wire#w1
   // the same network as SCL:
   "IN".HOOTER_RESET := "HOOTER_RESET" OR "HMI".HOOTER_RESET;
END_REGION

REGION Network 3: POWER_FAIL
   RUNG wire#powerrail
      I_Contact( "POWER_FAIL" )
      Coil( "IN".POWER_FAIL )
   END_RUNG
   // the same network as SCL:
   "IN".POWER_FAIL := NOT "POWER_FAIL";
END_REGION

REGION Network 4: "AIR_PRESSURE_SWITCH"
   RUNG wire#powerrail
      I_Contact( "AIR PRESSURE FAIL" )
      Coil( "IN".AIR_SWITCH )
   END_RUNG
   // the same network as SCL:
   "IN".AIR_SWITCH := NOT "AIR PRESSURE FAIL";
END_REGION

REGION Network 5: "CENTRIFUGAL_PUMP-1_TRIP"
   RUNG wire#powerrail
      Contact( "CENTRIFUGAL_PUMP-1_TRIP_(FWD)" )
      Coil( "IN"."PUMP-1_TRIP" )
   END_RUNG
   // the same network as SCL:
   "IN"."PUMP-1_TRIP" := "CENTRIFUGAL_PUMP-1_TRIP_(FWD)";
END_REGION

REGION Network 6: "CENTRIFUGAL_PUMP-2_TRIP"
   RUNG wire#powerrail
      Contact( "CENTRIFUGAL_PUMP-2_TRIP_(RET)" )
      Coil( "IN"."PUMP-2_TRIP" )
   END_RUNG
   // the same network as SCL:
   "IN"."PUMP-2_TRIP" := "CENTRIFUGAL_PUMP-2_TRIP_(RET)";
END_REGION

REGION Network 7: "FLOW SWITCH-1"
   RUNG wire#powerrail
      Contact( "FLOW SWITCH-1" )
      Coil( "IN".LSW_FWD_PUMP )
   END_RUNG
   // the same network as SCL:
   "IN".LSW_FWD_PUMP := "FLOW SWITCH-1";
END_REGION

REGION Network 8: "FLOW SWITCH-2"
   RUNG wire#powerrail
      Contact( "FLOW SWITCH-2" )
      Coil( "IN".LSW_RET_PUMP )
   END_RUNG
   // the same network as SCL:
   "IN".LSW_RET_PUMP := "FLOW SWITCH-2";
END_REGION

REGION Network 9: "LEVEL_SWITCH-1" SOFT WATER
   RUNG wire#powerrail
      Contact( "LEVEL_SWITCH-1" )
      Coil( "IN".SWT_HL )
   END_RUNG
   RUNG wire#powerrail
      I_Contact( "LEVEL_SWITCH-1" )
      Coil( "IN".SWT_LL )
   END_RUNG
   // the same network as SCL:
   "IN".SWT_HL := "LEVEL_SWITCH-1";
   "IN".SWT_LL := NOT "LEVEL_SWITCH-1";
END_REGION

REGION Network 10: "LEVEL_SWITCH-2" PW
   RUNG wire#powerrail
      Contact( "LEVEL_SWITCH-2" )
      Coil( "IN".PWT_HL )
   END_RUNG
   RUNG wire#powerrail
      I_Contact( "LEVEL_SWITCH-2" )
      Coil( "IN".PWT_LL )
   END_RUNG
   // the same network as SCL:
   "IN".PWT_HL := "LEVEL_SWITCH-2";
   "IN".PWT_LL := NOT "LEVEL_SWITCH-2";
END_REGION

REGION Network 11: "LEVEL_SWITCH-3" ALKALI
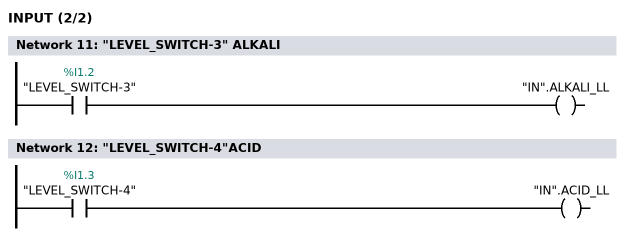
   RUNG wire#powerrail
      Contact( "LEVEL_SWITCH-3" )
      Coil( "IN".ALKALI_LL )
   END_RUNG
   // the same network as SCL:
   "IN".ALKALI_LL := "LEVEL_SWITCH-3";
END_REGION

REGION Network 12: "LEVEL_SWITCH-4"ACID
   RUNG wire#powerrail
      Contact( "LEVEL_SWITCH-4" )
      Coil( "IN".ACID_LL )
   END_RUNG
   // the same network as SCL:
   "IN".ACID_LL := "LEVEL_SWITCH-4";
END_REGION
END_FUNCTION

FUNCTION "MODE" : Void   // FC3, LAD
{ S7_Optimized_Access := 'TRUE' }
// stored: SetENOAutomatically false
   VAR_TEMP   // added for the SCL form of the ladder/FBD networks
      _w1 : Bool;
   END_VAR
BEGIN

REGION Network 1: MANUAL_MODE_SELECTION
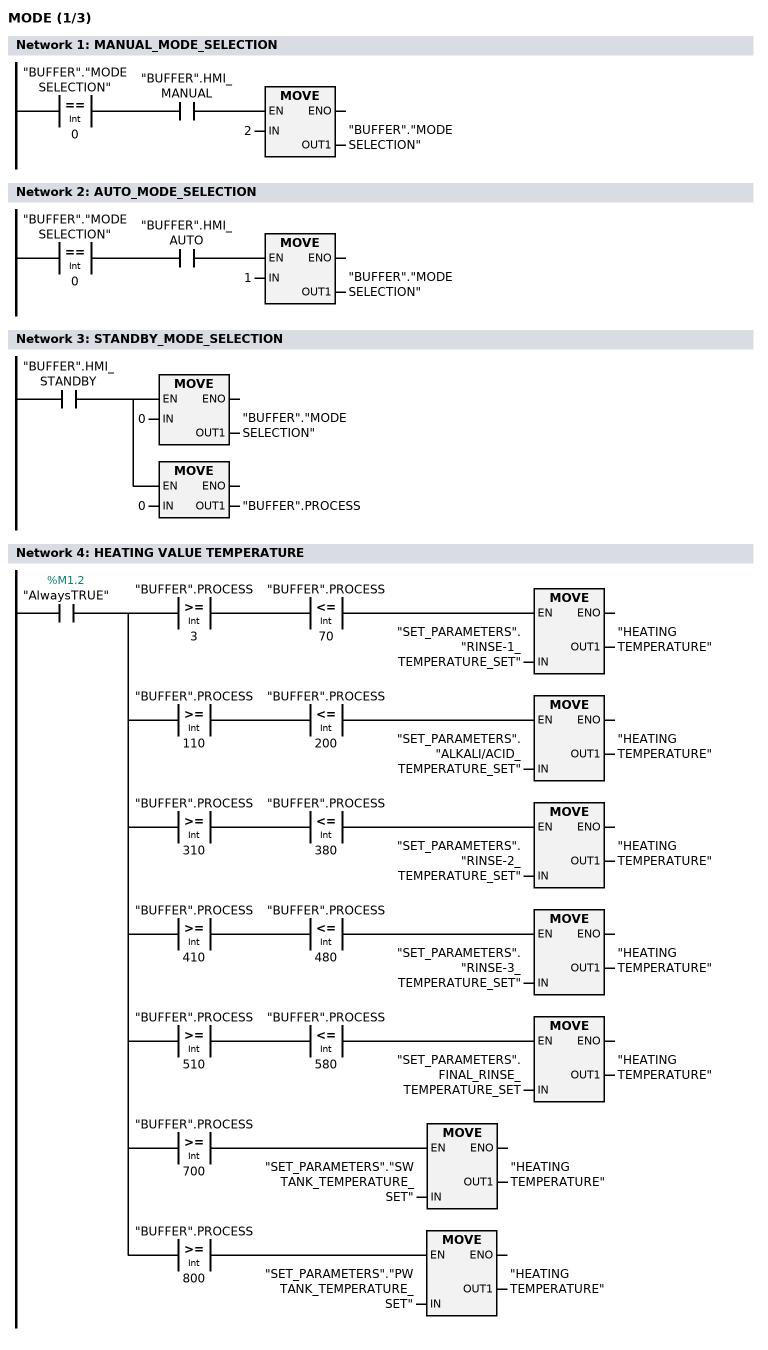
   RUNG wire#powerrail
      { S7_Templates := "SrcType := Int" } EQ_Contact(in1 := "BUFFER"."MODE SELECTION", in2 := 0)
      Contact( "BUFFER".HMI_MANUAL )
      Move(in := 2, out1 => "BUFFER"."MODE SELECTION")
   END_RUNG
   // the same network as SCL:
   IF ("BUFFER"."MODE SELECTION" = 0) AND "BUFFER".HMI_MANUAL THEN "BUFFER"."MODE SELECTION" := 2; END_IF;
END_REGION

REGION Network 2: AUTO_MODE_SELECTION
   RUNG wire#powerrail
      { S7_Templates := "SrcType := Int" } EQ_Contact(in1 := "BUFFER"."MODE SELECTION", in2 := 0)
      Contact( "BUFFER".HMI_AUTO )
      Move(in := 1, out1 => "BUFFER"."MODE SELECTION")
   END_RUNG
   // the same network as SCL:
   IF ("BUFFER"."MODE SELECTION" = 0) AND "BUFFER".HMI_AUTO THEN "BUFFER"."MODE SELECTION" := 1; END_IF;
END_REGION

REGION Network 3: STANDBY_MODE_SELECTION
   RUNG wire#powerrail
      Contact( "BUFFER".HMI_STANDBY )
      wire#w1
      Move(in := 0, out1 => "BUFFER"."MODE SELECTION")
   END_RUNG
   RUNG wire#w1
      Move(in := 0, out1 => "BUFFER".PROCESS)
   END_RUNG
   // the same network as SCL:
   IF "BUFFER".HMI_STANDBY THEN
       "BUFFER"."MODE SELECTION" := 0;
       "BUFFER".PROCESS := 0;
   END_IF;
END_REGION

REGION Network 4: HEATING VALUE TEMPERATURE
   RUNG wire#powerrail
      Contact( "AlwaysTRUE" )
      wire#w1
      { S7_Templates := "SrcType := Int" } GE_Contact(in1 := "BUFFER".PROCESS, in2 := 3)
      { S7_Templates := "SrcType := Int" } LE_Contact(in1 := "BUFFER".PROCESS, in2 := 70)
      Move(in := "SET_PARAMETERS"."RINSE-1_TEMPERATURE_SET", out1 => "HEATING TEMPERATURE")
   END_RUNG
   RUNG wire#w1
      { S7_Templates := "SrcType := Int" } GE_Contact(in1 := "BUFFER".PROCESS, in2 := 110)
      { S7_Templates := "SrcType := Int" } LE_Contact(in1 := "BUFFER".PROCESS, in2 := 200)
      Move(in := "SET_PARAMETERS"."ALKALI/ACID_TEMPERATURE_SET", out1 => "HEATING TEMPERATURE")
   END_RUNG
   RUNG wire#w1
      { S7_Templates := "SrcType := Int" } GE_Contact(in1 := "BUFFER".PROCESS, in2 := 310)
      { S7_Templates := "SrcType := Int" } LE_Contact(in1 := "BUFFER".PROCESS, in2 := 380)
      Move(in := "SET_PARAMETERS"."RINSE-2_TEMPERATURE_SET", out1 => "HEATING TEMPERATURE")
   END_RUNG
   RUNG wire#w1
      { S7_Templates := "SrcType := Int" } GE_Contact(in1 := "BUFFER".PROCESS, in2 := 410)
      { S7_Templates := "SrcType := Int" } LE_Contact(in1 := "BUFFER".PROCESS, in2 := 480)
      Move(in := "SET_PARAMETERS"."RINSE-3_TEMPERATURE_SET", out1 => "HEATING TEMPERATURE")
   END_RUNG
   RUNG wire#w1
      { S7_Templates := "SrcType := Int" } GE_Contact(in1 := "BUFFER".PROCESS, in2 := 510)
      { S7_Templates := "SrcType := Int" } LE_Contact(in1 := "BUFFER".PROCESS, in2 := 580)
      Move(in := "SET_PARAMETERS".FINAL_RINSE_TEMPERATURE_SET, out1 => "HEATING TEMPERATURE")
   END_RUNG
   RUNG wire#w1
      { S7_Templates := "SrcType := Int" } GE_Contact(in1 := "BUFFER".PROCESS, in2 := 700)
      Move(in := "SET_PARAMETERS"."SW TANK_TEMPERATURE_SET", out1 => "HEATING TEMPERATURE")
   END_RUNG
   RUNG wire#w1
      { S7_Templates := "SrcType := Int" } GE_Contact(in1 := "BUFFER".PROCESS, in2 := 800)
      Move(in := "SET_PARAMETERS"."PW TANK_TEMPERATURE_SET", out1 => "HEATING TEMPERATURE")
   END_RUNG
   // the same network as SCL:
   IF "AlwaysTRUE" AND ("BUFFER".PROCESS >= 3) AND ("BUFFER".PROCESS <= 70) THEN
       "HEATING TEMPERATURE" := "SET_PARAMETERS"."RINSE-1_TEMPERATURE_SET";
   END_IF;
   IF "AlwaysTRUE" AND ("BUFFER".PROCESS >= 110) AND ("BUFFER".PROCESS <= 200) THEN
       "HEATING TEMPERATURE" := "SET_PARAMETERS"."ALKALI/ACID_TEMPERATURE_SET";
   END_IF;
   IF "AlwaysTRUE" AND ("BUFFER".PROCESS >= 310) AND ("BUFFER".PROCESS <= 380) THEN
       "HEATING TEMPERATURE" := "SET_PARAMETERS"."RINSE-2_TEMPERATURE_SET";
   END_IF;
   IF "AlwaysTRUE" AND ("BUFFER".PROCESS >= 410) AND ("BUFFER".PROCESS <= 480) THEN
       "HEATING TEMPERATURE" := "SET_PARAMETERS"."RINSE-3_TEMPERATURE_SET";
   END_IF;
   IF "AlwaysTRUE" AND ("BUFFER".PROCESS >= 510) AND ("BUFFER".PROCESS <= 580) THEN
       "HEATING TEMPERATURE" := "SET_PARAMETERS".FINAL_RINSE_TEMPERATURE_SET;
   END_IF;
   IF "AlwaysTRUE" AND ("BUFFER".PROCESS >= 700) THEN
       "HEATING TEMPERATURE" := "SET_PARAMETERS"."SW TANK_TEMPERATURE_SET";
   END_IF;
   IF "AlwaysTRUE" AND ("BUFFER".PROCESS >= 800) THEN
       "HEATING TEMPERATURE" := "SET_PARAMETERS"."PW TANK_TEMPERATURE_SET";
   END_IF;
END_REGION

REGION Network 5: HEATING HYSTERSIS
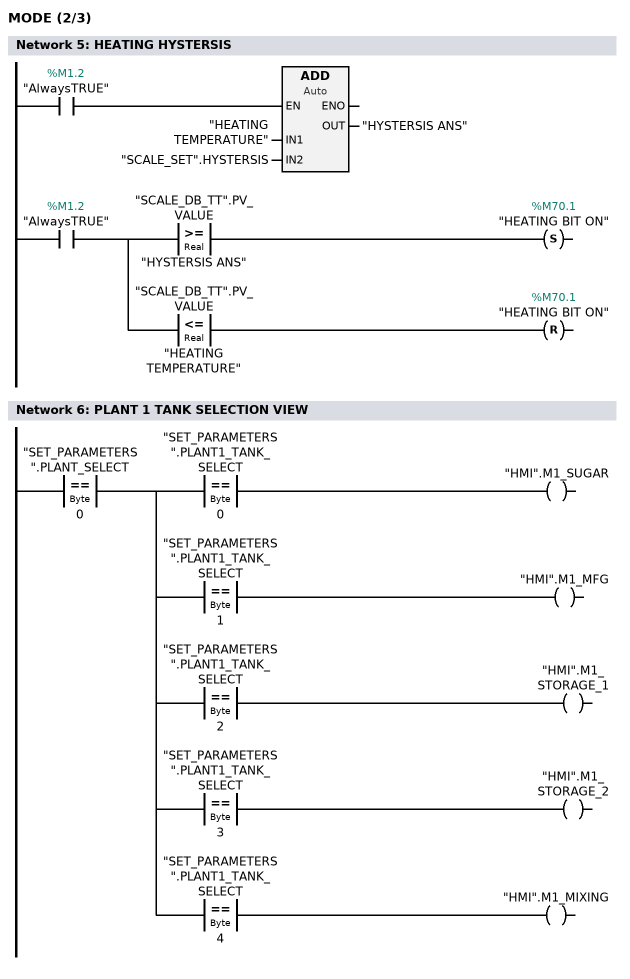
   RUNG wire#powerrail
      Contact( "AlwaysTRUE" )
      Add(in1 := "HEATING TEMPERATURE", in2 := "SCALE_SET".HYSTERSIS, out => "HYSTERSIS ANS")
   END_RUNG
   RUNG wire#powerrail
      Contact( "AlwaysTRUE" )
      wire#w1
      { S7_Templates := "SrcType := Real" } GE_Contact(in1 := "SCALE_DB_TT".PV_VALUE, in2 := "HYSTERSIS ANS")
      S_Coil( "HEATING BIT ON" )
   END_RUNG
   RUNG wire#w1
      { S7_Templates := "SrcType := Real" } LE_Contact(in1 := "SCALE_DB_TT".PV_VALUE, in2 := "HEATING TEMPERATURE")
      R_Coil( "HEATING BIT ON" )
   END_RUNG
   // the same network as SCL:
   IF "AlwaysTRUE" THEN "HYSTERSIS ANS" := "HEATING TEMPERATURE" + "SCALE_SET".HYSTERSIS; END_IF;
   IF "AlwaysTRUE" AND ("SCALE_DB_TT".PV_VALUE >= "HYSTERSIS ANS") THEN "HEATING BIT ON" := TRUE; END_IF;
   IF "AlwaysTRUE" AND ("SCALE_DB_TT".PV_VALUE <= "HEATING TEMPERATURE") THEN
       "HEATING BIT ON" := FALSE;
   END_IF;
END_REGION

REGION Network 6: PLANT 1 TANK SELECTION VIEW
   RUNG wire#powerrail
      { S7_Templates := "SrcType := Byte" } EQ_Contact(in1 := "SET_PARAMETERS".PLANT_SELECT, in2 := 0)
      wire#w1
      { S7_Templates := "SrcType := Byte" } EQ_Contact(in1 := "SET_PARAMETERS".PLANT1_TANK_SELECT, in2 := 0)
      Coil( "HMI".M1_SUGAR )
   END_RUNG
   RUNG wire#w1
      { S7_Templates := "SrcType := Byte" } EQ_Contact(in1 := "SET_PARAMETERS".PLANT1_TANK_SELECT, in2 := 1)
      Coil( "HMI".M1_MFG )
   END_RUNG
   RUNG wire#w1
      { S7_Templates := "SrcType := Byte" } EQ_Contact(in1 := "SET_PARAMETERS".PLANT1_TANK_SELECT, in2 := 2)
      Coil( "HMI".M1_STORAGE_1 )
   END_RUNG
   RUNG wire#w1
      { S7_Templates := "SrcType := Byte" } EQ_Contact(in1 := "SET_PARAMETERS".PLANT1_TANK_SELECT, in2 := 3)
      Coil( "HMI".M1_STORAGE_2 )
   END_RUNG
   RUNG wire#w1
      { S7_Templates := "SrcType := Byte" } EQ_Contact(in1 := "SET_PARAMETERS".PLANT1_TANK_SELECT, in2 := 4)
      Coil( "HMI".M1_MIXING )
   END_RUNG
   // the same network as SCL:
   #_w1 := "SET_PARAMETERS".PLANT_SELECT = 0;
   "HMI".M1_SUGAR := #_w1 AND ("SET_PARAMETERS".PLANT1_TANK_SELECT = 0);
   "HMI".M1_MFG := #_w1 AND ("SET_PARAMETERS".PLANT1_TANK_SELECT = 1);
   "HMI".M1_STORAGE_1 := #_w1 AND ("SET_PARAMETERS".PLANT1_TANK_SELECT = 2);
   "HMI".M1_STORAGE_2 := #_w1 AND ("SET_PARAMETERS".PLANT1_TANK_SELECT = 3);
   "HMI".M1_MIXING := #_w1 AND ("SET_PARAMETERS".PLANT1_TANK_SELECT = 4);
END_REGION

REGION Network 7: PLANT 2 TANK SELECTION VIEW
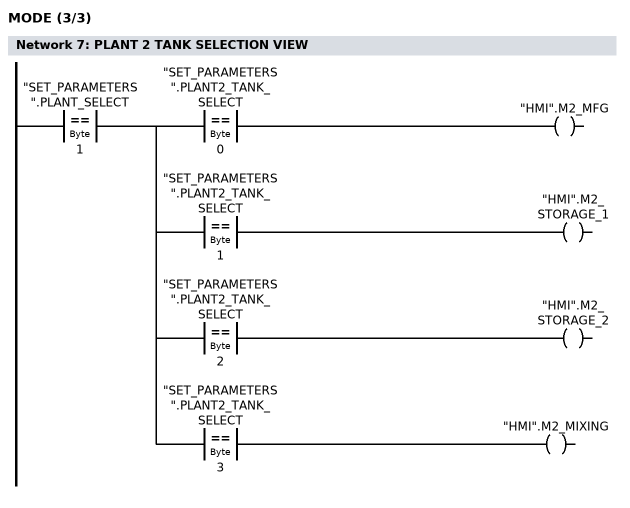
   RUNG wire#powerrail
      { S7_Templates := "SrcType := Byte" } EQ_Contact(in1 := "SET_PARAMETERS".PLANT_SELECT, in2 := 1)
      wire#w1
      { S7_Templates := "SrcType := Byte" } EQ_Contact(in1 := "SET_PARAMETERS".PLANT2_TANK_SELECT, in2 := 0)
      Coil( "HMI".M2_MFG )
   END_RUNG
   RUNG wire#w1
      { S7_Templates := "SrcType := Byte" } EQ_Contact(in1 := "SET_PARAMETERS".PLANT2_TANK_SELECT, in2 := 1)
      Coil( "HMI".M2_STORAGE_1 )
   END_RUNG
   RUNG wire#w1
      { S7_Templates := "SrcType := Byte" } EQ_Contact(in1 := "SET_PARAMETERS".PLANT2_TANK_SELECT, in2 := 2)
      Coil( "HMI".M2_STORAGE_2 )
   END_RUNG
   RUNG wire#w1
      { S7_Templates := "SrcType := Byte" } EQ_Contact(in1 := "SET_PARAMETERS".PLANT2_TANK_SELECT, in2 := 3)
      Coil( "HMI".M2_MIXING )
   END_RUNG
   // the same network as SCL:
   #_w1 := "SET_PARAMETERS".PLANT_SELECT = 1;
   "HMI".M2_MFG := #_w1 AND ("SET_PARAMETERS".PLANT2_TANK_SELECT = 0);
   "HMI".M2_STORAGE_1 := #_w1 AND ("SET_PARAMETERS".PLANT2_TANK_SELECT = 1);
   "HMI".M2_STORAGE_2 := #_w1 AND ("SET_PARAMETERS".PLANT2_TANK_SELECT = 2);
   "HMI".M2_MIXING := #_w1 AND ("SET_PARAMETERS".PLANT2_TANK_SELECT = 3);
END_REGION
END_FUNCTION

FUNCTION "AUTO_LOGIC_FOR_CIP_TANK" : Void   // FC13, LAD
{ S7_Optimized_Access := 'TRUE' }
// stored: SetENOAutomatically false
   VAR_TEMP   // added for the SCL form of the ladder/FBD networks
      _w1 : Bool;
      _w2 : Bool;
      _w3 : Bool;
      _w4 : Bool;
   END_VAR
BEGIN

REGION Network 1: START
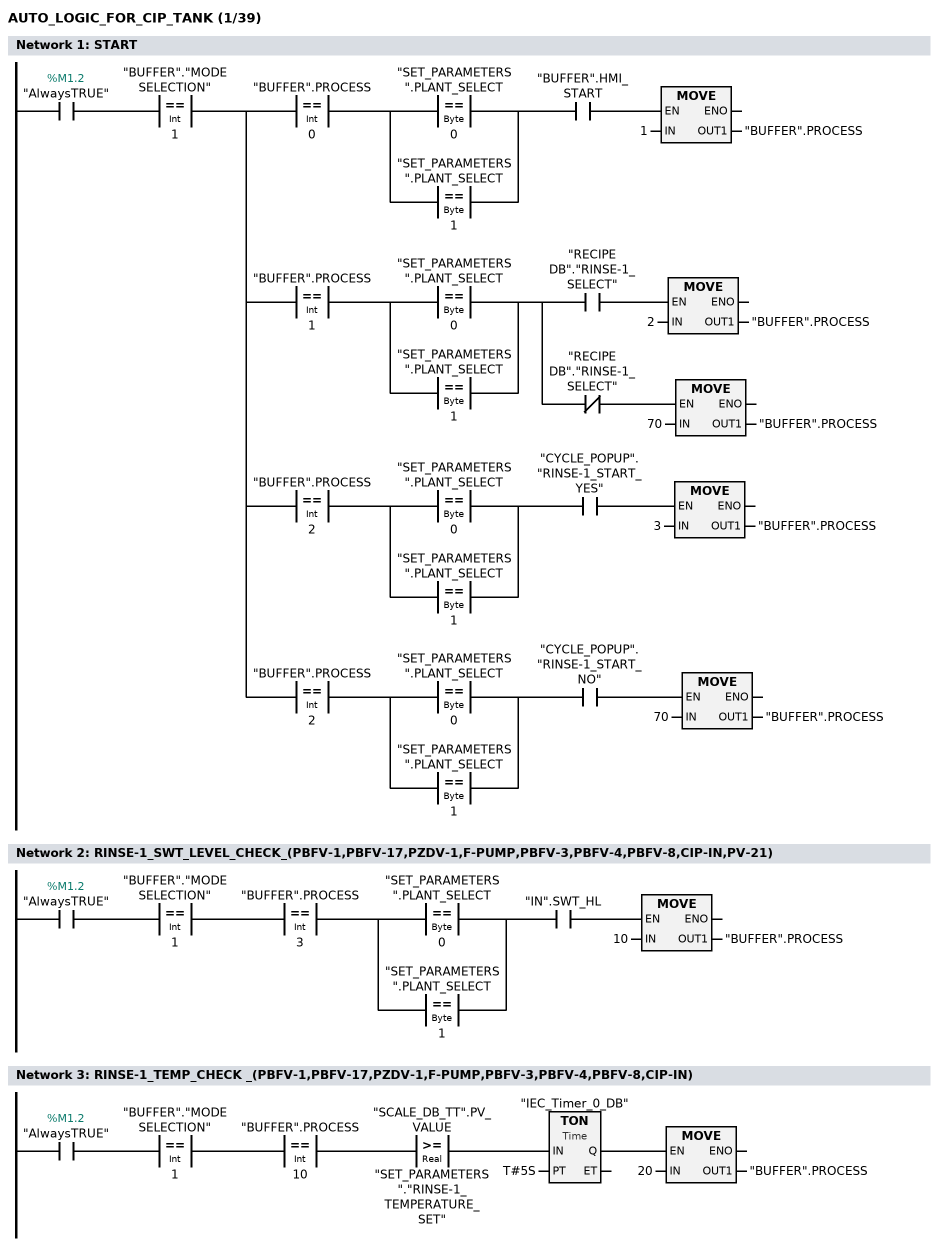
   RUNG wire#powerrail
      Contact( "AlwaysTRUE" )
      { S7_Templates := "SrcType := Int" } EQ_Contact(in1 := "BUFFER"."MODE SELECTION", in2 := 1)
      wire#w1
      { S7_Templates := "SrcType := Int" } EQ_Contact(in1 := "BUFFER".PROCESS, in2 := 0)
      wire#w2
      { S7_Templates := "SrcType := Byte" } EQ_Contact(in1 := "SET_PARAMETERS".PLANT_SELECT, in2 := 0)
      wire#w3
      Contact( "BUFFER".HMI_START )
      Move(in := 1, out1 => "BUFFER".PROCESS)
   END_RUNG
   RUNG wire#w2
      { S7_Templates := "SrcType := Byte" } EQ_Contact(in1 := "SET_PARAMETERS".PLANT_SELECT, in2 := 1)
   END_RUNG wire#w3
   RUNG wire#w1
      { S7_Templates := "SrcType := Int" } EQ_Contact(in1 := "BUFFER".PROCESS, in2 := 1)
      wire#w4
      { S7_Templates := "SrcType := Byte" } EQ_Contact(in1 := "SET_PARAMETERS".PLANT_SELECT, in2 := 0)
      wire#w5
      Contact( "RECIPE DB"."RINSE-1_SELECT" )
      Move(in := 2, out1 => "BUFFER".PROCESS)
   END_RUNG
   RUNG wire#w4
      { S7_Templates := "SrcType := Byte" } EQ_Contact(in1 := "SET_PARAMETERS".PLANT_SELECT, in2 := 1)
   END_RUNG wire#w5
   RUNG wire#w5
      I_Contact( "RECIPE DB"."RINSE-1_SELECT" )
      Move(in := 70, out1 => "BUFFER".PROCESS)
   END_RUNG
   RUNG wire#w1
      { S7_Templates := "SrcType := Int" } EQ_Contact(in1 := "BUFFER".PROCESS, in2 := 2)
      wire#w6
      { S7_Templates := "SrcType := Byte" } EQ_Contact(in1 := "SET_PARAMETERS".PLANT_SELECT, in2 := 0)
      wire#w7
      Contact( "CYCLE_POPUP"."RINSE-1_START_YES" )
      Move(in := 3, out1 => "BUFFER".PROCESS)
   END_RUNG
   RUNG wire#w6
      { S7_Templates := "SrcType := Byte" } EQ_Contact(in1 := "SET_PARAMETERS".PLANT_SELECT, in2 := 1)
   END_RUNG wire#w7
   RUNG wire#w1
      { S7_Templates := "SrcType := Int" } EQ_Contact(in1 := "BUFFER".PROCESS, in2 := 2)
      wire#w8
      { S7_Templates := "SrcType := Byte" } EQ_Contact(in1 := "SET_PARAMETERS".PLANT_SELECT, in2 := 0)
      wire#w9
      Contact( "CYCLE_POPUP"."RINSE-1_START_NO" )
      Move(in := 70, out1 => "BUFFER".PROCESS)
   END_RUNG
   RUNG wire#w8
      { S7_Templates := "SrcType := Byte" } EQ_Contact(in1 := "SET_PARAMETERS".PLANT_SELECT, in2 := 1)
   END_RUNG wire#w9
   // the same network as SCL:
   #_w1 := "AlwaysTRUE" AND ("BUFFER"."MODE SELECTION" = 1);
   IF #_w1 AND ("BUFFER".PROCESS = 0) AND (("SET_PARAMETERS".PLANT_SELECT = 0) OR ("SET_PARAMETERS".PLANT_SELECT = 1)) AND "BUFFER".HMI_START THEN
       "BUFFER".PROCESS := 1;
   END_IF;
   #_w2 := #_w1 AND ("BUFFER".PROCESS = 1) AND (("SET_PARAMETERS".PLANT_SELECT = 0) OR ("SET_PARAMETERS".PLANT_SELECT = 1));
   IF #_w2 AND "RECIPE DB"."RINSE-1_SELECT" THEN "BUFFER".PROCESS := 2; END_IF;
   IF #_w2 AND NOT "RECIPE DB"."RINSE-1_SELECT" THEN "BUFFER".PROCESS := 70; END_IF;
   IF #_w1 AND ("BUFFER".PROCESS = 2) AND (("SET_PARAMETERS".PLANT_SELECT = 0) OR ("SET_PARAMETERS".PLANT_SELECT = 1)) AND "CYCLE_POPUP"."RINSE-1_START_YES" THEN
       "BUFFER".PROCESS := 3;
   END_IF;
   IF #_w1 AND ("BUFFER".PROCESS = 2) AND (("SET_PARAMETERS".PLANT_SELECT = 0) OR ("SET_PARAMETERS".PLANT_SELECT = 1)) AND "CYCLE_POPUP"."RINSE-1_START_NO" THEN
       "BUFFER".PROCESS := 70;
   END_IF;
END_REGION

REGION Network 2: RINSE-1_SWT_LEVEL_CHECK_(PBFV-1,PBFV-17,PZDV-1,F-PUMP,PBFV-3,PBFV-4,PBFV-8,CIP-IN,PV-21)
   RUNG wire#powerrail
      Contact( "AlwaysTRUE" )
      { S7_Templates := "SrcType := Int" } EQ_Contact(in1 := "BUFFER"."MODE SELECTION", in2 := 1)
      { S7_Templates := "SrcType := Int" } EQ_Contact(in1 := "BUFFER".PROCESS, in2 := 3)
      wire#w1
      { S7_Templates := "SrcType := Byte" } EQ_Contact(in1 := "SET_PARAMETERS".PLANT_SELECT, in2 := 0)
      wire#w2
      Contact( "IN".SWT_HL )
      Move(in := 10, out1 => "BUFFER".PROCESS)
   END_RUNG
   RUNG wire#w1
      { S7_Templates := "SrcType := Byte" } EQ_Contact(in1 := "SET_PARAMETERS".PLANT_SELECT, in2 := 1)
   END_RUNG wire#w2
   // the same network as SCL:
   IF "AlwaysTRUE" AND ("BUFFER"."MODE SELECTION" = 1) AND ("BUFFER".PROCESS = 3) AND (("SET_PARAMETERS".PLANT_SELECT = 0) OR ("SET_PARAMETERS".PLANT_SELECT = 1)) AND "IN".SWT_HL THEN
       "BUFFER".PROCESS := 10;
   END_IF;
END_REGION

REGION Network 3: RINSE-1_TEMP_CHECK _(PBFV-1,PBFV-17,PZDV-1,F-PUMP,PBFV-3,PBFV-4,PBFV-8,CIP-IN)
   RUNG wire#powerrail
      Contact( "AlwaysTRUE" )
      { S7_Templates := "SrcType := Int" } EQ_Contact(in1 := "BUFFER"."MODE SELECTION", in2 := 1)
      { S7_Templates := "SrcType := Int" } EQ_Contact(in1 := "BUFFER".PROCESS, in2 := 10)
      { S7_Templates := "SrcType := Real" } GE_Contact(in1 := "SCALE_DB_TT".PV_VALUE, in2 := "SET_PARAMETERS"."RINSE-1_TEMPERATURE_SET")
      { S7_Templates := "time_type := Time" } "IEC_Timer_0_DB".TON(pt := T#5S, et =>)
      Move(in := 20, out1 => "BUFFER".PROCESS)
   END_RUNG
   // the same network as SCL:
   "IEC_Timer_0_DB".TON(IN := "AlwaysTRUE" AND ("BUFFER"."MODE SELECTION" = 1) AND ("BUFFER".PROCESS = 10) AND ("SCALE_DB_TT".PV_VALUE >= "SET_PARAMETERS"."RINSE-1_TEMPERATURE_SET"),
                        PT := T#5S);
   IF "IEC_Timer_0_DB".Q THEN "BUFFER".PROCESS := 20; END_IF;
END_REGION

REGION Network 4: RINSE-1_CLEANING_TIME_(PBFV-1,PBFV-17,PZDV-1,F-PUMP,PBFV-3,PBFV-4,PBFV-8,CIP-IN)
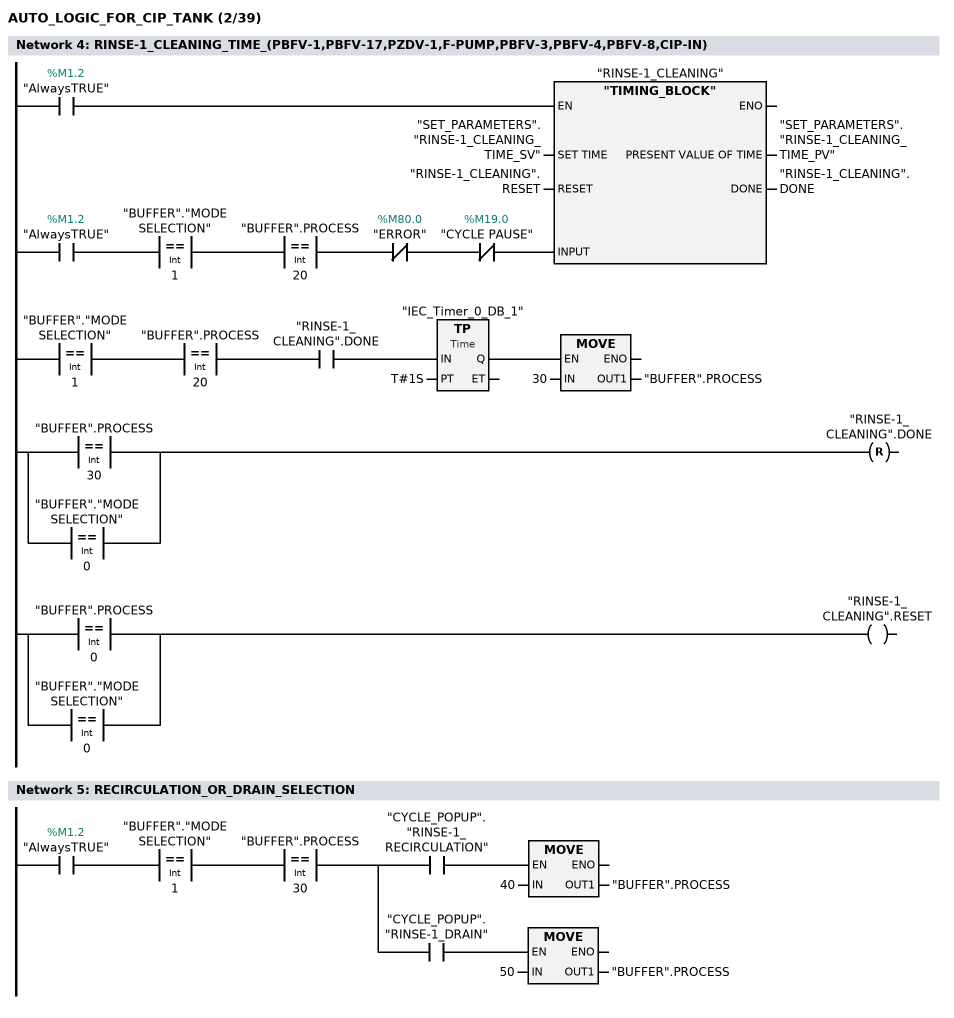
   RUNG wire#powerrail
      Contact( "AlwaysTRUE" )
      "RINSE-1_CLEANING"(INPUT := wire#w1, "SET TIME" := "SET_PARAMETERS"."RINSE-1_CLEANING_TIME_SV", RESET := "RINSE-1_CLEANING".RESET, "PRESENT VALUE OF TIME" => "SET_PARAMETERS"."RINSE-1_CLEANING_TIME_PV", DONE => "RINSE-1_CLEANING".DONE)
   END_RUNG
   RUNG wire#powerrail
      Contact( "AlwaysTRUE" )
      { S7_Templates := "SrcType := Int" } EQ_Contact(in1 := "BUFFER"."MODE SELECTION", in2 := 1)
      { S7_Templates := "SrcType := Int" } EQ_Contact(in1 := "BUFFER".PROCESS, in2 := 20)
      I_Contact( "ERROR" )
      I_Contact( "CYCLE PAUSE" )
   END_RUNG wire#w1
   RUNG wire#powerrail
      { S7_Templates := "SrcType := Int" } EQ_Contact(in1 := "BUFFER"."MODE SELECTION", in2 := 1)
      { S7_Templates := "SrcType := Int" } EQ_Contact(in1 := "BUFFER".PROCESS, in2 := 20)
      Contact( "RINSE-1_CLEANING".DONE )
      { S7_Templates := "time_type := Time" } "IEC_Timer_0_DB_1".TP(pt := T#1S, et =>)
      Move(in := 30, out1 => "BUFFER".PROCESS)
   END_RUNG
   RUNG wire#powerrail
      { S7_Templates := "SrcType := Int" } EQ_Contact(in1 := "BUFFER".PROCESS, in2 := 30)
      wire#w2
      R_Coil( "RINSE-1_CLEANING".DONE )
   END_RUNG
   RUNG wire#powerrail
      { S7_Templates := "SrcType := Int" } EQ_Contact(in1 := "BUFFER"."MODE SELECTION", in2 := 0)
   END_RUNG wire#w2
   RUNG wire#powerrail
      { S7_Templates := "SrcType := Int" } EQ_Contact(in1 := "BUFFER".PROCESS, in2 := 0)
      wire#w3
      Coil( "RINSE-1_CLEANING".RESET )
   END_RUNG
   RUNG wire#powerrail
      { S7_Templates := "SrcType := Int" } EQ_Contact(in1 := "BUFFER"."MODE SELECTION", in2 := 0)
   END_RUNG wire#w3
   // the same network as SCL:
   IF "AlwaysTRUE" THEN
       "RINSE-1_CLEANING"("SET TIME" := "SET_PARAMETERS"."RINSE-1_CLEANING_TIME_SV",   // "TIMING_BLOCK"
                          RESET := "RINSE-1_CLEANING".RESET,
                          INPUT := "AlwaysTRUE" AND ("BUFFER"."MODE SELECTION" = 1) AND ("BUFFER".PROCESS = 20) AND NOT "ERROR" AND NOT "CYCLE PAUSE",
                          "PRESENT VALUE OF TIME" => "SET_PARAMETERS"."RINSE-1_CLEANING_TIME_PV",
                          DONE => "RINSE-1_CLEANING".DONE);
   END_IF;
   "IEC_Timer_0_DB_1".TP(IN := ("BUFFER"."MODE SELECTION" = 1) AND ("BUFFER".PROCESS = 20) AND "RINSE-1_CLEANING".DONE,
                         PT := T#1S);
   IF "IEC_Timer_0_DB_1".Q THEN "BUFFER".PROCESS := 30; END_IF;
   IF ("BUFFER".PROCESS = 30) OR ("BUFFER"."MODE SELECTION" = 0) THEN
       "RINSE-1_CLEANING".DONE := FALSE;
   END_IF;
   "RINSE-1_CLEANING".RESET := ("BUFFER".PROCESS = 0) OR ("BUFFER"."MODE SELECTION" = 0);
END_REGION

REGION Network 5: RECIRCULATION_OR_DRAIN_SELECTION
   RUNG wire#powerrail
      Contact( "AlwaysTRUE" )
      { S7_Templates := "SrcType := Int" } EQ_Contact(in1 := "BUFFER"."MODE SELECTION", in2 := 1)
      { S7_Templates := "SrcType := Int" } EQ_Contact(in1 := "BUFFER".PROCESS, in2 := 30)
      wire#w1
      Contact( "CYCLE_POPUP"."RINSE-1_RECIRCULATION" )
      Move(in := 40, out1 => "BUFFER".PROCESS)
   END_RUNG
   RUNG wire#w1
      Contact( "CYCLE_POPUP"."RINSE-1_DRAIN" )
      Move(in := 50, out1 => "BUFFER".PROCESS)
   END_RUNG
   // the same network as SCL:
   #_w1 := "AlwaysTRUE" AND ("BUFFER"."MODE SELECTION" = 1) AND ("BUFFER".PROCESS = 30);
   IF #_w1 AND "CYCLE_POPUP"."RINSE-1_RECIRCULATION" THEN "BUFFER".PROCESS := 40; END_IF;
   IF #_w1 AND "CYCLE_POPUP"."RINSE-1_DRAIN" THEN "BUFFER".PROCESS := 50; END_IF;
END_REGION

REGION Network 6: RINSE-1_RECIRCULATION_TIME_(CIP-OUT,R-PUMP,PBFV-6,PBFV-8,CIP-IN)
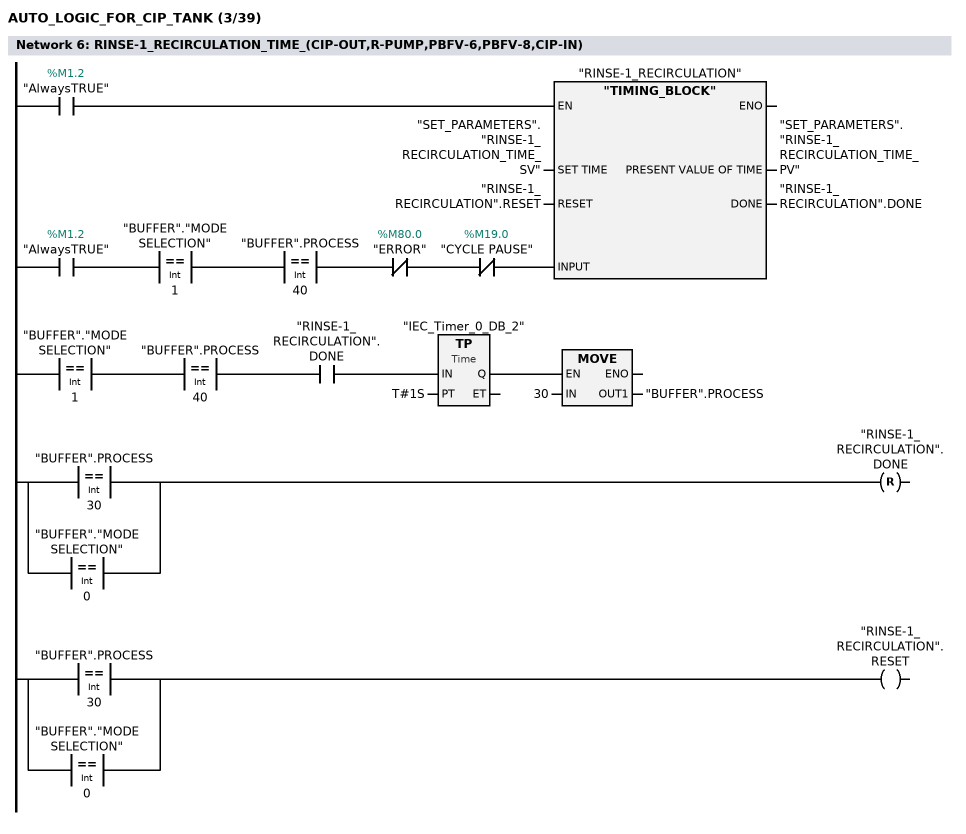
   RUNG wire#powerrail
      Contact( "AlwaysTRUE" )
      "RINSE-1_RECIRCULATION"(INPUT := wire#w1, "SET TIME" := "SET_PARAMETERS"."RINSE-1_RECIRCULATION_TIME_SV", RESET := "RINSE-1_RECIRCULATION".RESET, "PRESENT VALUE OF TIME" => "SET_PARAMETERS"."RINSE-1_RECIRCULATION_TIME_PV", DONE => "RINSE-1_RECIRCULATION".DONE)
   END_RUNG
   RUNG wire#powerrail
      Contact( "AlwaysTRUE" )
      { S7_Templates := "SrcType := Int" } EQ_Contact(in1 := "BUFFER"."MODE SELECTION", in2 := 1)
      { S7_Templates := "SrcType := Int" } EQ_Contact(in1 := "BUFFER".PROCESS, in2 := 40)
      I_Contact( "ERROR" )
      I_Contact( "CYCLE PAUSE" )
   END_RUNG wire#w1
   RUNG wire#powerrail
      { S7_Templates := "SrcType := Int" } EQ_Contact(in1 := "BUFFER"."MODE SELECTION", in2 := 1)
      { S7_Templates := "SrcType := Int" } EQ_Contact(in1 := "BUFFER".PROCESS, in2 := 40)
      Contact( "RINSE-1_RECIRCULATION".DONE )
      { S7_Templates := "time_type := Time" } "IEC_Timer_0_DB_2".TP(pt := T#1S, et =>)
      Move(in := 30, out1 => "BUFFER".PROCESS)
   END_RUNG
   RUNG wire#powerrail
      { S7_Templates := "SrcType := Int" } EQ_Contact(in1 := "BUFFER".PROCESS, in2 := 30)
      wire#w2
      R_Coil( "RINSE-1_RECIRCULATION".DONE )
   END_RUNG
   RUNG wire#powerrail
      { S7_Templates := "SrcType := Int" } EQ_Contact(in1 := "BUFFER"."MODE SELECTION", in2 := 0)
   END_RUNG wire#w2
   RUNG wire#powerrail
      { S7_Templates := "SrcType := Int" } EQ_Contact(in1 := "BUFFER".PROCESS, in2 := 30)
      wire#w3
      Coil( "RINSE-1_RECIRCULATION".RESET )
   END_RUNG
   RUNG wire#powerrail
      { S7_Templates := "SrcType := Int" } EQ_Contact(in1 := "BUFFER"."MODE SELECTION", in2 := 0)
   END_RUNG wire#w3
   // the same network as SCL:
   IF "AlwaysTRUE" THEN
       "RINSE-1_RECIRCULATION"("SET TIME" := "SET_PARAMETERS"."RINSE-1_RECIRCULATION_TIME_SV",   // "TIMING_BLOCK"
                               RESET := "RINSE-1_RECIRCULATION".RESET,
                               INPUT := "AlwaysTRUE" AND ("BUFFER"."MODE SELECTION" = 1) AND ("BUFFER".PROCESS = 40) AND NOT "ERROR" AND NOT "CYCLE PAUSE",
                               "PRESENT VALUE OF TIME" => "SET_PARAMETERS"."RINSE-1_RECIRCULATION_TIME_PV",
                               DONE => "RINSE-1_RECIRCULATION".DONE);
   END_IF;
   "IEC_Timer_0_DB_2".TP(IN := ("BUFFER"."MODE SELECTION" = 1) AND ("BUFFER".PROCESS = 40) AND "RINSE-1_RECIRCULATION".DONE,
                         PT := T#1S);
   IF "IEC_Timer_0_DB_2".Q THEN "BUFFER".PROCESS := 30; END_IF;
   IF ("BUFFER".PROCESS = 30) OR ("BUFFER"."MODE SELECTION" = 0) THEN
       "RINSE-1_RECIRCULATION".DONE := FALSE;
   END_IF;
   "RINSE-1_RECIRCULATION".RESET := ("BUFFER".PROCESS = 30) OR ("BUFFER"."MODE SELECTION" = 0);
END_REGION

REGION Network 7: RINSE-1_DRAIN_TIME_(CIP-OUT,R_PUMP,PBFV-11)
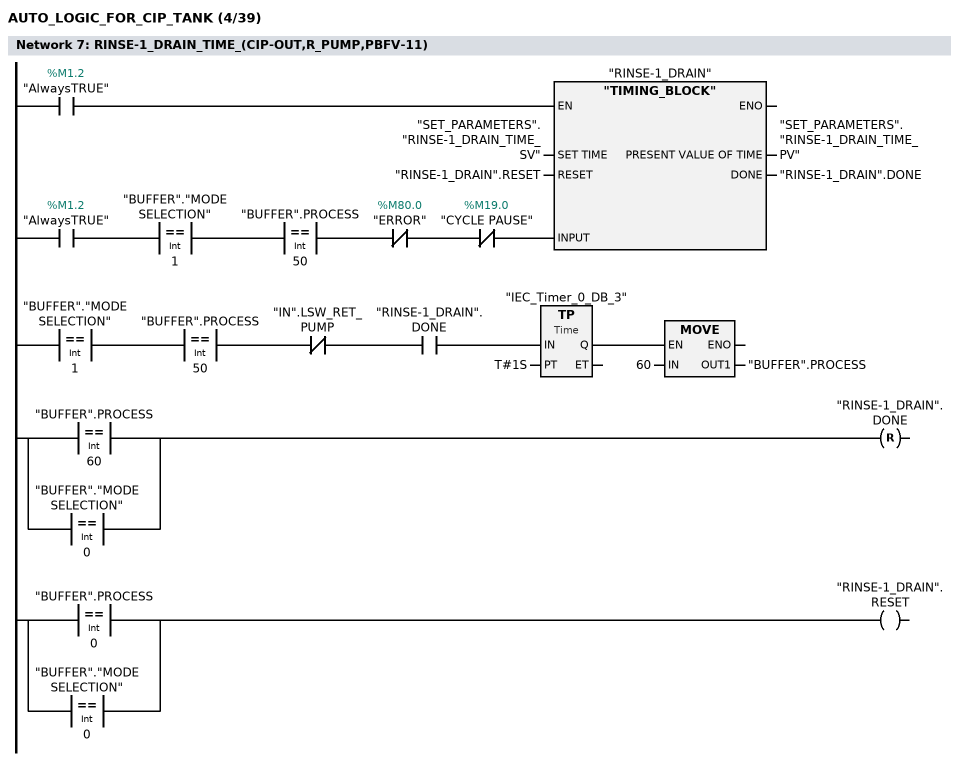
   RUNG wire#powerrail
      Contact( "AlwaysTRUE" )
      "RINSE-1_DRAIN"(INPUT := wire#w1, "SET TIME" := "SET_PARAMETERS"."RINSE-1_DRAIN_TIME_SV", RESET := "RINSE-1_DRAIN".RESET, "PRESENT VALUE OF TIME" => "SET_PARAMETERS"."RINSE-1_DRAIN_TIME_PV", DONE => "RINSE-1_DRAIN".DONE)
   END_RUNG
   RUNG wire#powerrail
      Contact( "AlwaysTRUE" )
      { S7_Templates := "SrcType := Int" } EQ_Contact(in1 := "BUFFER"."MODE SELECTION", in2 := 1)
      { S7_Templates := "SrcType := Int" } EQ_Contact(in1 := "BUFFER".PROCESS, in2 := 50)
      I_Contact( "ERROR" )
      I_Contact( "CYCLE PAUSE" )
   END_RUNG wire#w1
   RUNG wire#powerrail
      { S7_Templates := "SrcType := Int" } EQ_Contact(in1 := "BUFFER"."MODE SELECTION", in2 := 1)
      { S7_Templates := "SrcType := Int" } EQ_Contact(in1 := "BUFFER".PROCESS, in2 := 50)
      I_Contact( "IN".LSW_RET_PUMP )
      Contact( "RINSE-1_DRAIN".DONE )
      { S7_Templates := "time_type := Time" } "IEC_Timer_0_DB_3".TP(pt := T#1S, et =>)
      Move(in := 60, out1 => "BUFFER".PROCESS)
   END_RUNG
   RUNG wire#powerrail
      { S7_Templates := "SrcType := Int" } EQ_Contact(in1 := "BUFFER".PROCESS, in2 := 60)
      wire#w2
      R_Coil( "RINSE-1_DRAIN".DONE )
   END_RUNG
   RUNG wire#powerrail
      { S7_Templates := "SrcType := Int" } EQ_Contact(in1 := "BUFFER"."MODE SELECTION", in2 := 0)
   END_RUNG wire#w2
   RUNG wire#powerrail
      { S7_Templates := "SrcType := Int" } EQ_Contact(in1 := "BUFFER".PROCESS, in2 := 0)
      wire#w3
      Coil( "RINSE-1_DRAIN".RESET )
   END_RUNG
   RUNG wire#powerrail
      { S7_Templates := "SrcType := Int" } EQ_Contact(in1 := "BUFFER"."MODE SELECTION", in2 := 0)
   END_RUNG wire#w3
   // the same network as SCL:
   IF "AlwaysTRUE" THEN
       "RINSE-1_DRAIN"("SET TIME" := "SET_PARAMETERS"."RINSE-1_DRAIN_TIME_SV",   // "TIMING_BLOCK"
                       RESET := "RINSE-1_DRAIN".RESET,
                       INPUT := "AlwaysTRUE" AND ("BUFFER"."MODE SELECTION" = 1) AND ("BUFFER".PROCESS = 50) AND NOT "ERROR" AND NOT "CYCLE PAUSE",
                       "PRESENT VALUE OF TIME" => "SET_PARAMETERS"."RINSE-1_DRAIN_TIME_PV",
                       DONE => "RINSE-1_DRAIN".DONE);
   END_IF;
   "IEC_Timer_0_DB_3".TP(IN := ("BUFFER"."MODE SELECTION" = 1) AND ("BUFFER".PROCESS = 50) AND NOT "IN".LSW_RET_PUMP AND "RINSE-1_DRAIN".DONE,
                         PT := T#1S);
   IF "IEC_Timer_0_DB_3".Q THEN "BUFFER".PROCESS := 60; END_IF;
   IF ("BUFFER".PROCESS = 60) OR ("BUFFER"."MODE SELECTION" = 0) THEN "RINSE-1_DRAIN".DONE := FALSE; END_IF;
   "RINSE-1_DRAIN".RESET := ("BUFFER".PROCESS = 0) OR ("BUFFER"."MODE SELECTION" = 0);
END_REGION

REGION Network 8: RINSE-1_PUMP_CHASING_TIME(PBFV-12,PBFV13)
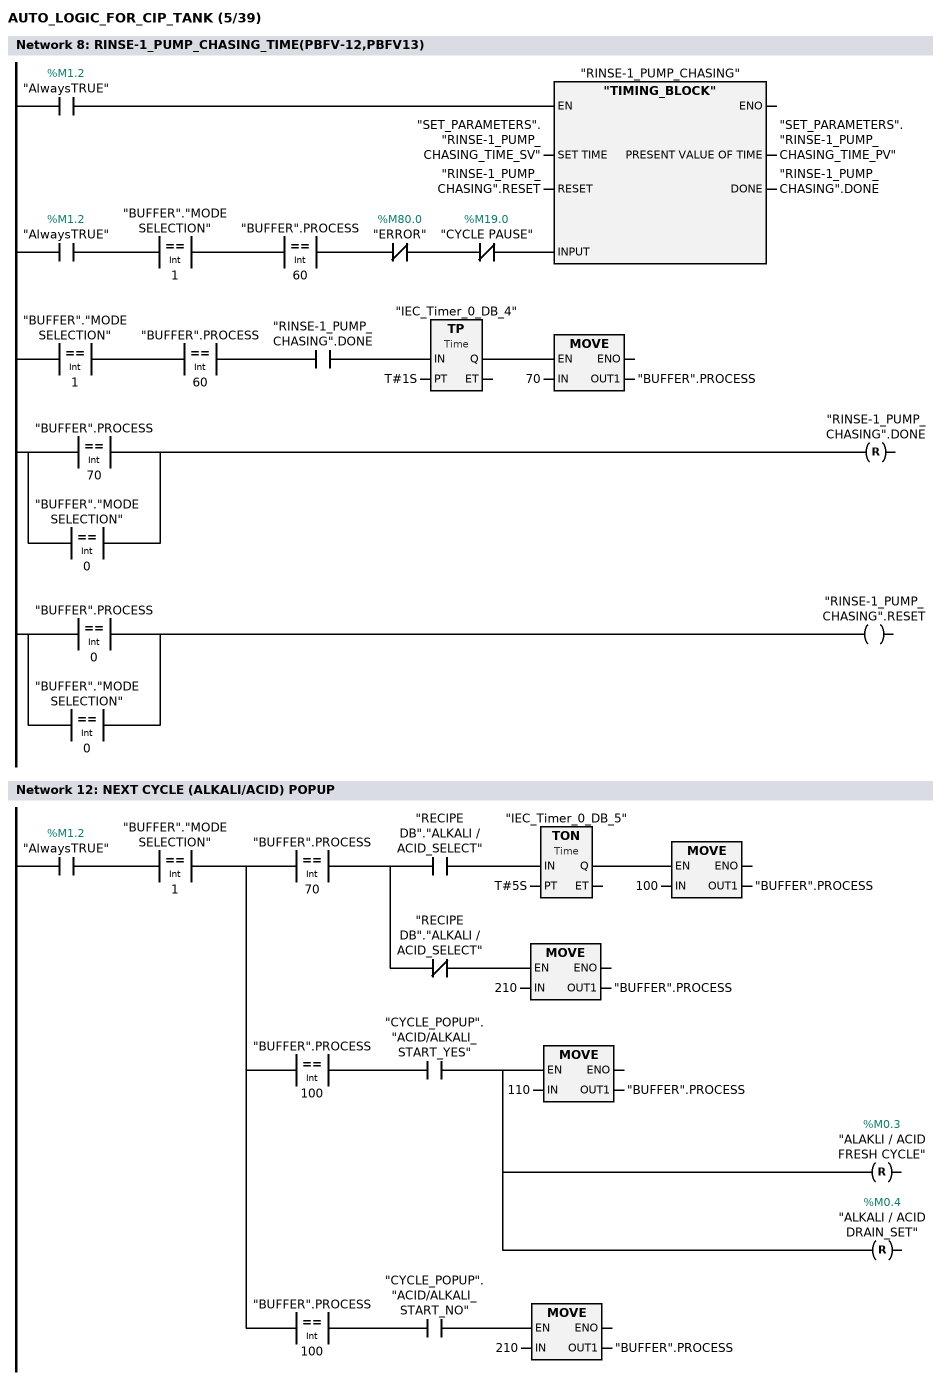
   RUNG wire#powerrail
      Contact( "AlwaysTRUE" )
      "RINSE-1_PUMP_CHASING"(INPUT := wire#w1, "SET TIME" := "SET_PARAMETERS"."RINSE-1_PUMP_CHASING_TIME_SV", RESET := "RINSE-1_PUMP_CHASING".RESET, "PRESENT VALUE OF TIME" => "SET_PARAMETERS"."RINSE-1_PUMP_CHASING_TIME_PV", DONE => "RINSE-1_PUMP_CHASING".DONE)
   END_RUNG
   RUNG wire#powerrail
      Contact( "AlwaysTRUE" )
      { S7_Templates := "SrcType := Int" } EQ_Contact(in1 := "BUFFER"."MODE SELECTION", in2 := 1)
      { S7_Templates := "SrcType := Int" } EQ_Contact(in1 := "BUFFER".PROCESS, in2 := 60)
      I_Contact( "ERROR" )
      I_Contact( "CYCLE PAUSE" )
   END_RUNG wire#w1
   RUNG wire#powerrail
      { S7_Templates := "SrcType := Int" } EQ_Contact(in1 := "BUFFER"."MODE SELECTION", in2 := 1)
      { S7_Templates := "SrcType := Int" } EQ_Contact(in1 := "BUFFER".PROCESS, in2 := 60)
      Contact( "RINSE-1_PUMP_CHASING".DONE )
      { S7_Templates := "time_type := Time" } "IEC_Timer_0_DB_4".TP(pt := T#1S, et =>)
      Move(in := 70, out1 => "BUFFER".PROCESS)
   END_RUNG
   RUNG wire#powerrail
      { S7_Templates := "SrcType := Int" } EQ_Contact(in1 := "BUFFER".PROCESS, in2 := 70)
      wire#w2
      R_Coil( "RINSE-1_PUMP_CHASING".DONE )
   END_RUNG
   RUNG wire#powerrail
      { S7_Templates := "SrcType := Int" } EQ_Contact(in1 := "BUFFER"."MODE SELECTION", in2 := 0)
   END_RUNG wire#w2
   RUNG wire#powerrail
      { S7_Templates := "SrcType := Int" } EQ_Contact(in1 := "BUFFER".PROCESS, in2 := 0)
      wire#w3
      Coil( "RINSE-1_PUMP_CHASING".RESET )
   END_RUNG
   RUNG wire#powerrail
      { S7_Templates := "SrcType := Int" } EQ_Contact(in1 := "BUFFER"."MODE SELECTION", in2 := 0)
   END_RUNG wire#w3
   // the same network as SCL:
   IF "AlwaysTRUE" THEN
       "RINSE-1_PUMP_CHASING"("SET TIME" := "SET_PARAMETERS"."RINSE-1_PUMP_CHASING_TIME_SV",   // "TIMING_BLOCK"
                              RESET := "RINSE-1_PUMP_CHASING".RESET,
                              INPUT := "AlwaysTRUE" AND ("BUFFER"."MODE SELECTION" = 1) AND ("BUFFER".PROCESS = 60) AND NOT "ERROR" AND NOT "CYCLE PAUSE",
                              "PRESENT VALUE OF TIME" => "SET_PARAMETERS"."RINSE-1_PUMP_CHASING_TIME_PV",
                              DONE => "RINSE-1_PUMP_CHASING".DONE);
   END_IF;
   "IEC_Timer_0_DB_4".TP(IN := ("BUFFER"."MODE SELECTION" = 1) AND ("BUFFER".PROCESS = 60) AND "RINSE-1_PUMP_CHASING".DONE,
                         PT := T#1S);
   IF "IEC_Timer_0_DB_4".Q THEN "BUFFER".PROCESS := 70; END_IF;
   IF ("BUFFER".PROCESS = 70) OR ("BUFFER"."MODE SELECTION" = 0) THEN
       "RINSE-1_PUMP_CHASING".DONE := FALSE;
   END_IF;
   "RINSE-1_PUMP_CHASING".RESET := ("BUFFER".PROCESS = 0) OR ("BUFFER"."MODE SELECTION" = 0);
END_REGION

REGION Network 12: NEXT CYCLE (ALKALI/ACID) POPUP
   RUNG wire#powerrail
      Contact( "AlwaysTRUE" )
      { S7_Templates := "SrcType := Int" } EQ_Contact(in1 := "BUFFER"."MODE SELECTION", in2 := 1)
      wire#w1
      { S7_Templates := "SrcType := Int" } EQ_Contact(in1 := "BUFFER".PROCESS, in2 := 70)
      wire#w2
      Contact( "RECIPE DB"."ALKALI / ACID_SELECT" )
      { S7_Templates := "time_type := Time" } "IEC_Timer_0_DB_5".TON(pt := T#5S, et =>)
      Move(in := 100, out1 => "BUFFER".PROCESS)
   END_RUNG
   RUNG wire#w2
      I_Contact( "RECIPE DB"."ALKALI / ACID_SELECT" )
      Move(in := 210, out1 => "BUFFER".PROCESS)
   END_RUNG
   RUNG wire#w1
      { S7_Templates := "SrcType := Int" } EQ_Contact(in1 := "BUFFER".PROCESS, in2 := 100)
      Contact( "CYCLE_POPUP"."ACID/ALKALI_START_YES" )
      wire#w3
      Move(in := 110, out1 => "BUFFER".PROCESS)
   END_RUNG
   RUNG wire#w3
      R_Coil( "ALAKLI / ACID FRESH CYCLE" )
   END_RUNG
   RUNG wire#w3
      R_Coil( "ALKALI / ACID DRAIN_SET" )
   END_RUNG
   RUNG wire#w1
      { S7_Templates := "SrcType := Int" } EQ_Contact(in1 := "BUFFER".PROCESS, in2 := 100)
      Contact( "CYCLE_POPUP"."ACID/ALKALI_START_NO" )
      Move(in := 210, out1 => "BUFFER".PROCESS)
   END_RUNG
   // the same network as SCL:
   #_w1 := "AlwaysTRUE" AND ("BUFFER"."MODE SELECTION" = 1);
   #_w2 := #_w1 AND ("BUFFER".PROCESS = 70);
   "IEC_Timer_0_DB_5".TON(IN := #_w2 AND "RECIPE DB"."ALKALI / ACID_SELECT", PT := T#5S);
   IF "IEC_Timer_0_DB_5".Q THEN "BUFFER".PROCESS := 100; END_IF;
   IF #_w2 AND NOT "RECIPE DB"."ALKALI / ACID_SELECT" THEN "BUFFER".PROCESS := 210; END_IF;
   #_w3 := #_w1 AND ("BUFFER".PROCESS = 100) AND "CYCLE_POPUP"."ACID/ALKALI_START_YES";
   IF #_w3 THEN
       "BUFFER".PROCESS := 110;
       "ALAKLI / ACID FRESH CYCLE" := FALSE;
       "ALKALI / ACID DRAIN_SET" := FALSE;
   END_IF;
   IF #_w1 AND ("BUFFER".PROCESS = 100) AND "CYCLE_POPUP"."ACID/ALKALI_START_NO" THEN
       "BUFFER".PROCESS := 210;
   END_IF;
END_REGION

REGION Network 13: SWT_LEVEL_CHECK(PBFV-17) POPUP + temperature cleaing
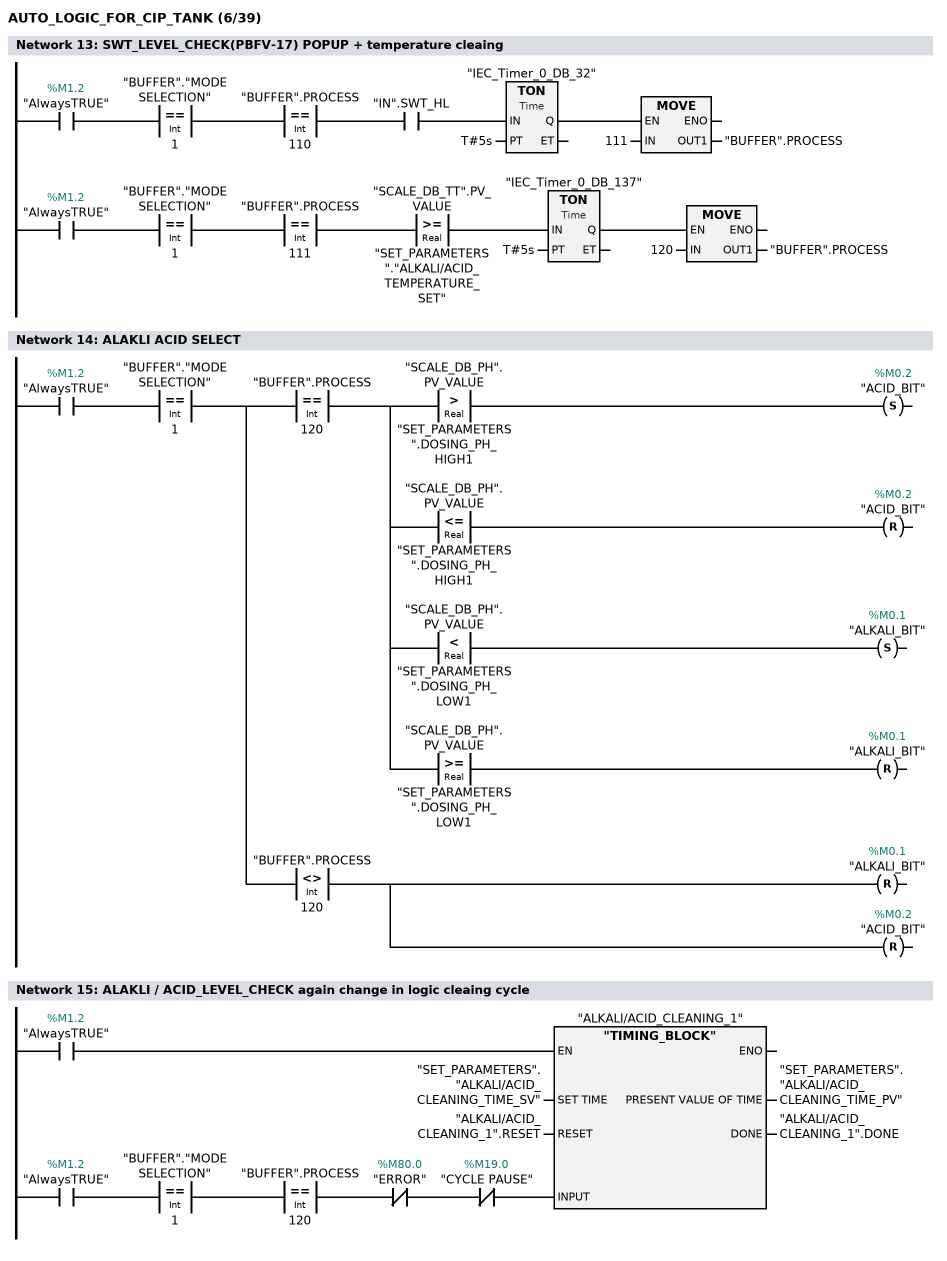
   RUNG wire#powerrail
      Contact( "AlwaysTRUE" )
      { S7_Templates := "SrcType := Int" } EQ_Contact(in1 := "BUFFER"."MODE SELECTION", in2 := 1)
      { S7_Templates := "SrcType := Int" } EQ_Contact(in1 := "BUFFER".PROCESS, in2 := 110)
      Contact( "IN".SWT_HL )
      { S7_Templates := "time_type := Time" } "IEC_Timer_0_DB_32".TON(pt := T#5s, et =>)
      Move(in := 111, out1 => "BUFFER".PROCESS)
   END_RUNG
   RUNG wire#powerrail
      Contact( "AlwaysTRUE" )
      { S7_Templates := "SrcType := Int" } EQ_Contact(in1 := "BUFFER"."MODE SELECTION", in2 := 1)
      { S7_Templates := "SrcType := Int" } EQ_Contact(in1 := "BUFFER".PROCESS, in2 := 111)
      { S7_Templates := "SrcType := Real" } GE_Contact(in1 := "SCALE_DB_TT".PV_VALUE, in2 := "SET_PARAMETERS"."ALKALI/ACID_TEMPERATURE_SET")
      { S7_Templates := "time_type := Time" } "IEC_Timer_0_DB_137".TON(pt := T#5s, et =>)
      Move(in := 120, out1 => "BUFFER".PROCESS)
   END_RUNG
   // the same network as SCL:
   "IEC_Timer_0_DB_32".TON(IN := "AlwaysTRUE" AND ("BUFFER"."MODE SELECTION" = 1) AND ("BUFFER".PROCESS = 110) AND "IN".SWT_HL,
                           PT := T#5s);
   IF "IEC_Timer_0_DB_32".Q THEN "BUFFER".PROCESS := 111; END_IF;
   "IEC_Timer_0_DB_137".TON(IN := "AlwaysTRUE" AND ("BUFFER"."MODE SELECTION" = 1) AND ("BUFFER".PROCESS = 111) AND ("SCALE_DB_TT".PV_VALUE >= "SET_PARAMETERS"."ALKALI/ACID_TEMPERATURE_SET"),
                           PT := T#5s);
   IF "IEC_Timer_0_DB_137".Q THEN "BUFFER".PROCESS := 120; END_IF;
END_REGION

REGION Network 14: ALAKLI ACID SELECT
   RUNG wire#powerrail
      Contact( "AlwaysTRUE" )
      { S7_Templates := "SrcType := Int" } EQ_Contact(in1 := "BUFFER"."MODE SELECTION", in2 := 1)
      wire#w1
      { S7_Templates := "SrcType := Int" } EQ_Contact(in1 := "BUFFER".PROCESS, in2 := 120)
      wire#w2
      { S7_Templates := "SrcType := Real" } GT_Contact(in1 := "SCALE_DB_PH".PV_VALUE, in2 := "SET_PARAMETERS".DOSING_PH_HIGH1)
      S_Coil( "ACID_BIT" )
   END_RUNG
   RUNG wire#w2
      { S7_Templates := "SrcType := Real" } LE_Contact(in1 := "SCALE_DB_PH".PV_VALUE, in2 := "SET_PARAMETERS".DOSING_PH_HIGH1)
      R_Coil( "ACID_BIT" )
   END_RUNG
   RUNG wire#w2
      { S7_Templates := "SrcType := Real" } LT_Contact(in1 := "SCALE_DB_PH".PV_VALUE, in2 := "SET_PARAMETERS".DOSING_PH_LOW1)
      S_Coil( "ALKALI_BIT" )
   END_RUNG
   RUNG wire#w2
      { S7_Templates := "SrcType := Real" } GE_Contact(in1 := "SCALE_DB_PH".PV_VALUE, in2 := "SET_PARAMETERS".DOSING_PH_LOW1)
      R_Coil( "ALKALI_BIT" )
   END_RUNG
   RUNG wire#w1
      { S7_Templates := "SrcType := Int" } NE_Contact(in1 := "BUFFER".PROCESS, in2 := 120)
      wire#w3
      R_Coil( "ALKALI_BIT" )
   END_RUNG
   RUNG wire#w3
      R_Coil( "ACID_BIT" )
   END_RUNG
   // the same network as SCL:
   #_w1 := "AlwaysTRUE" AND ("BUFFER"."MODE SELECTION" = 1);
   #_w2 := #_w1 AND ("BUFFER".PROCESS = 120);
   IF #_w2 AND ("SCALE_DB_PH".PV_VALUE > "SET_PARAMETERS".DOSING_PH_HIGH1) THEN "ACID_BIT" := TRUE; END_IF;
   IF #_w2 AND ("SCALE_DB_PH".PV_VALUE <= "SET_PARAMETERS".DOSING_PH_HIGH1) THEN "ACID_BIT" := FALSE; END_IF;
   IF #_w2 AND ("SCALE_DB_PH".PV_VALUE < "SET_PARAMETERS".DOSING_PH_LOW1) THEN "ALKALI_BIT" := TRUE; END_IF;
   IF #_w2 AND ("SCALE_DB_PH".PV_VALUE >= "SET_PARAMETERS".DOSING_PH_LOW1) THEN
       "ALKALI_BIT" := FALSE;
   END_IF;
   IF #_w1 AND ("BUFFER".PROCESS <> 120) THEN
       "ALKALI_BIT" := FALSE;
       "ACID_BIT" := FALSE;
   END_IF;
END_REGION

REGION Network 15: ALAKLI / ACID_LEVEL_CHECK again change in logic cleaing cycle
   RUNG wire#powerrail
      Contact( "AlwaysTRUE" )
      "ALKALI/ACID_CLEANING_1"(INPUT := wire#w1, "SET TIME" := "SET_PARAMETERS"."ALKALI/ACID_CLEANING_TIME_SV", RESET := "ALKALI/ACID_CLEANING_1".RESET, "PRESENT VALUE OF TIME" => "SET_PARAMETERS"."ALKALI/ACID_CLEANING_TIME_PV", DONE => "ALKALI/ACID_CLEANING_1".DONE)
   END_RUNG
   RUNG wire#powerrail
      Contact( "AlwaysTRUE" )
      { S7_Templates := "SrcType := Int" } EQ_Contact(in1 := "BUFFER"."MODE SELECTION", in2 := 1)
      { S7_Templates := "SrcType := Int" } EQ_Contact(in1 := "BUFFER".PROCESS, in2 := 120)
      I_Contact( "ERROR" )
      I_Contact( "CYCLE PAUSE" )
   END_RUNG wire#w1
   // the same network as SCL:
   IF "AlwaysTRUE" THEN
       "ALKALI/ACID_CLEANING_1"("SET TIME" := "SET_PARAMETERS"."ALKALI/ACID_CLEANING_TIME_SV",   // "TIMING_BLOCK"
                               RESET := "ALKALI/ACID_CLEANING_1".RESET,
                               INPUT := "AlwaysTRUE" AND ("BUFFER"."MODE SELECTION" = 1) AND ("BUFFER".PROCESS = 120) AND NOT "ERROR" AND NOT "CYCLE PAUSE",
                               "PRESENT VALUE OF TIME" => "SET_PARAMETERS"."ALKALI/ACID_CLEANING_TIME_PV",
                               DONE => "ALKALI/ACID_CLEANING_1".DONE);
   END_IF;
END_REGION

REGION Network 16: use------------------
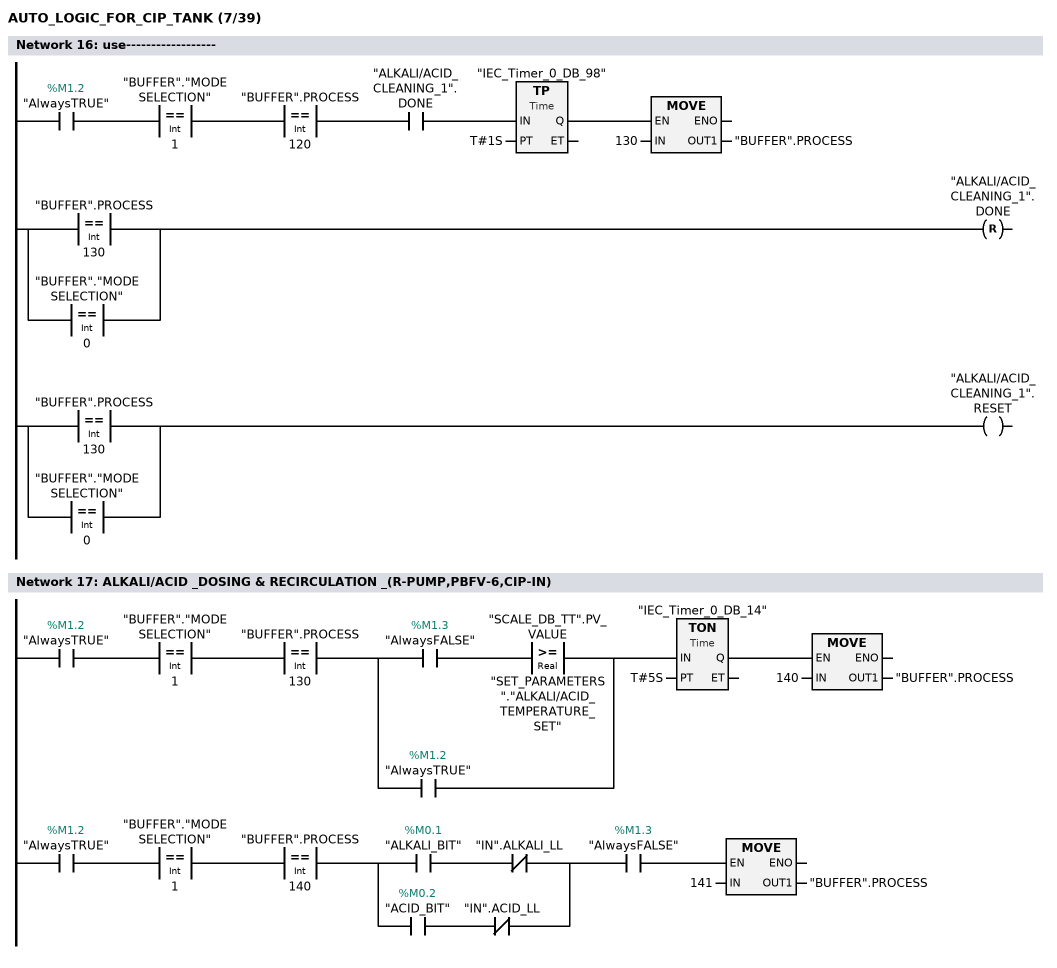
   RUNG wire#powerrail
      Contact( "AlwaysTRUE" )
      { S7_Templates := "SrcType := Int" } EQ_Contact(in1 := "BUFFER"."MODE SELECTION", in2 := 1)
      { S7_Templates := "SrcType := Int" } EQ_Contact(in1 := "BUFFER".PROCESS, in2 := 120)
      Contact( "ALKALI/ACID_CLEANING_1".DONE )
      { S7_Templates := "time_type := Time" } "IEC_Timer_0_DB_98".TP(pt := T#1S, et =>)
      Move(in := 130, out1 => "BUFFER".PROCESS)
   END_RUNG
   RUNG wire#powerrail
      { S7_Templates := "SrcType := Int" } EQ_Contact(in1 := "BUFFER".PROCESS, in2 := 130)
      wire#w1
      R_Coil( "ALKALI/ACID_CLEANING_1".DONE )
   END_RUNG
   RUNG wire#powerrail
      { S7_Templates := "SrcType := Int" } EQ_Contact(in1 := "BUFFER"."MODE SELECTION", in2 := 0)
   END_RUNG wire#w1
   RUNG wire#powerrail
      { S7_Templates := "SrcType := Int" } EQ_Contact(in1 := "BUFFER".PROCESS, in2 := 130)
      wire#w2
      Coil( "ALKALI/ACID_CLEANING_1".RESET )
   END_RUNG
   RUNG wire#powerrail
      { S7_Templates := "SrcType := Int" } EQ_Contact(in1 := "BUFFER"."MODE SELECTION", in2 := 0)
   END_RUNG wire#w2
   // the same network as SCL:
   "IEC_Timer_0_DB_98".TP(IN := "AlwaysTRUE" AND ("BUFFER"."MODE SELECTION" = 1) AND ("BUFFER".PROCESS = 120) AND "ALKALI/ACID_CLEANING_1".DONE,
                          PT := T#1S);
   IF "IEC_Timer_0_DB_98".Q THEN "BUFFER".PROCESS := 130; END_IF;
   IF ("BUFFER".PROCESS = 130) OR ("BUFFER"."MODE SELECTION" = 0) THEN
       "ALKALI/ACID_CLEANING_1".DONE := FALSE;
   END_IF;
   "ALKALI/ACID_CLEANING_1".RESET := ("BUFFER".PROCESS = 130) OR ("BUFFER"."MODE SELECTION" = 0);
END_REGION

REGION Network 17: ALKALI/ACID _DOSING & RECIRCULATION _(R-PUMP,PBFV-6,CIP-IN)
   RUNG wire#powerrail
      Contact( "AlwaysTRUE" )
      { S7_Templates := "SrcType := Int" } EQ_Contact(in1 := "BUFFER"."MODE SELECTION", in2 := 1)
      { S7_Templates := "SrcType := Int" } EQ_Contact(in1 := "BUFFER".PROCESS, in2 := 130)
      wire#w1
      Contact( "AlwaysFALSE" )
      { S7_Templates := "SrcType := Real" } GE_Contact(in1 := "SCALE_DB_TT".PV_VALUE, in2 := "SET_PARAMETERS"."ALKALI/ACID_TEMPERATURE_SET")
      wire#w2
      { S7_Templates := "time_type := Time" } "IEC_Timer_0_DB_14".TON(pt := T#5S, et =>)
      Move(in := 140, out1 => "BUFFER".PROCESS)
   END_RUNG
   RUNG wire#w1
      Contact( "AlwaysTRUE" )
   END_RUNG wire#w2
   RUNG wire#powerrail
      Contact( "AlwaysTRUE" )
      { S7_Templates := "SrcType := Int" } EQ_Contact(in1 := "BUFFER"."MODE SELECTION", in2 := 1)
      { S7_Templates := "SrcType := Int" } EQ_Contact(in1 := "BUFFER".PROCESS, in2 := 140)
      wire#w3
      Contact( "ALKALI_BIT" )
      I_Contact( "IN".ALKALI_LL )
      wire#w4
      Contact( "AlwaysFALSE" )
      Move(in := 141, out1 => "BUFFER".PROCESS)
   END_RUNG
   RUNG wire#w3
      Contact( "ACID_BIT" )
      I_Contact( "IN".ACID_LL )
   END_RUNG wire#w4
   // the same network as SCL:
   "IEC_Timer_0_DB_14".TON(IN := "AlwaysTRUE" AND ("BUFFER"."MODE SELECTION" = 1) AND ("BUFFER".PROCESS = 130) AND (("AlwaysFALSE" AND ("SCALE_DB_TT".PV_VALUE >= "SET_PARAMETERS"."ALKALI/ACID_TEMPERATURE_SET")) OR "AlwaysTRUE"),
                           PT := T#5S);
   IF "IEC_Timer_0_DB_14".Q THEN "BUFFER".PROCESS := 140; END_IF;
   IF "AlwaysTRUE" AND ("BUFFER"."MODE SELECTION" = 1) AND ("BUFFER".PROCESS = 140) AND (("ALKALI_BIT" AND NOT "IN".ALKALI_LL) OR ("ACID_BIT" AND NOT "IN".ACID_LL)) AND "AlwaysFALSE" THEN
       "BUFFER".PROCESS := 141;
   END_IF;
END_REGION

REGION Network 18: ALKALI/ACID_RECIRCULATION_TIME_(CIP-OUT,R-PUMP,PBFV-6,PBFV-8,CIP-IN)
   // recirculation + dosing
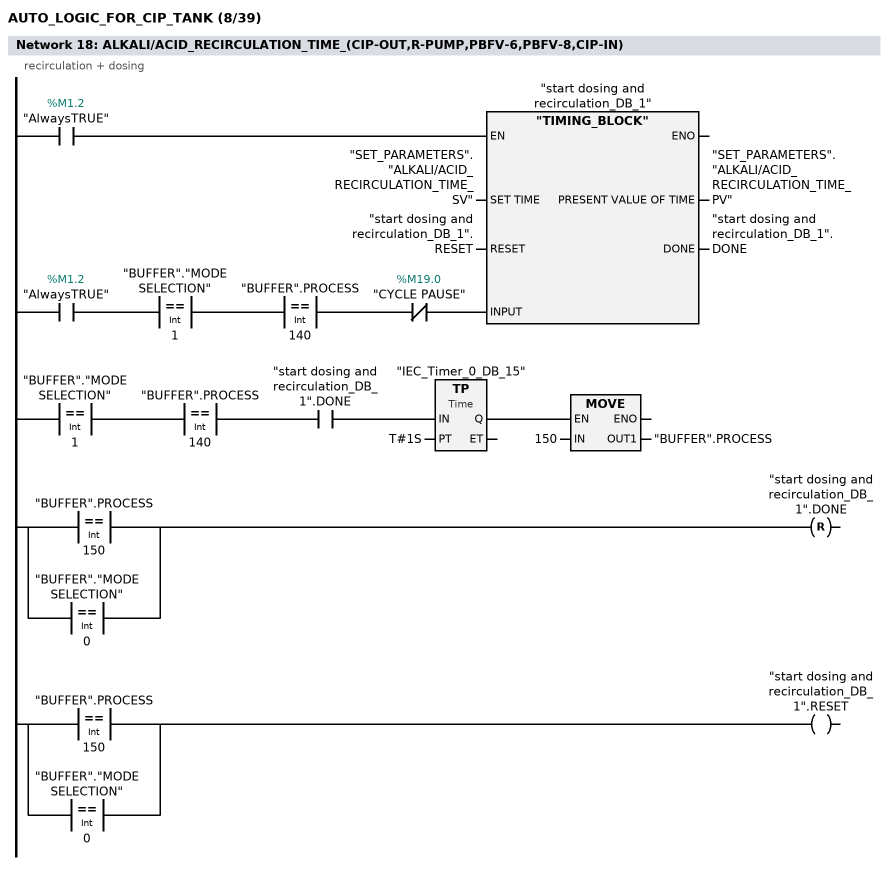
   RUNG wire#powerrail
      Contact( "AlwaysTRUE" )
      "start dosing and recirculation_DB_1"(INPUT := wire#w1, "SET TIME" := "SET_PARAMETERS"."ALKALI/ACID_RECIRCULATION_TIME_SV", RESET := "start dosing and recirculation_DB_1".RESET, "PRESENT VALUE OF TIME" => "SET_PARAMETERS"."ALKALI/ACID_RECIRCULATION_TIME_PV", DONE => "start dosing and recirculation_DB_1".DONE)
   END_RUNG
   RUNG wire#powerrail
      Contact( "AlwaysTRUE" )
      { S7_Templates := "SrcType := Int" } EQ_Contact(in1 := "BUFFER"."MODE SELECTION", in2 := 1)
      { S7_Templates := "SrcType := Int" } EQ_Contact(in1 := "BUFFER".PROCESS, in2 := 140)
      I_Contact( "CYCLE PAUSE" )
   END_RUNG wire#w1
   RUNG wire#powerrail
      { S7_Templates := "SrcType := Int" } EQ_Contact(in1 := "BUFFER"."MODE SELECTION", in2 := 1)
      { S7_Templates := "SrcType := Int" } EQ_Contact(in1 := "BUFFER".PROCESS, in2 := 140)
      Contact( "start dosing and recirculation_DB_1".DONE )
      { S7_Templates := "time_type := Time" } "IEC_Timer_0_DB_15".TP(pt := T#1S, et =>)
      Move(in := 150, out1 => "BUFFER".PROCESS)
   END_RUNG
   RUNG wire#powerrail
      { S7_Templates := "SrcType := Int" } EQ_Contact(in1 := "BUFFER".PROCESS, in2 := 150)
      wire#w2
      R_Coil( "start dosing and recirculation_DB_1".DONE )
   END_RUNG
   RUNG wire#powerrail
      { S7_Templates := "SrcType := Int" } EQ_Contact(in1 := "BUFFER"."MODE SELECTION", in2 := 0)
   END_RUNG wire#w2
   RUNG wire#powerrail
      { S7_Templates := "SrcType := Int" } EQ_Contact(in1 := "BUFFER".PROCESS, in2 := 150)
      wire#w3
      Coil( "start dosing and recirculation_DB_1".RESET )
   END_RUNG
   RUNG wire#powerrail
      { S7_Templates := "SrcType := Int" } EQ_Contact(in1 := "BUFFER"."MODE SELECTION", in2 := 0)
   END_RUNG wire#w3
   // the same network as SCL:
   IF "AlwaysTRUE" THEN
       "start dosing and recirculation_DB_1"("SET TIME" := "SET_PARAMETERS"."ALKALI/ACID_RECIRCULATION_TIME_SV",   // "TIMING_BLOCK"
                               RESET := "start dosing and recirculation_DB_1".RESET,
                               INPUT := "AlwaysTRUE" AND ("BUFFER"."MODE SELECTION" = 1) AND ("BUFFER".PROCESS = 140) AND NOT "CYCLE PAUSE",
                               "PRESENT VALUE OF TIME" => "SET_PARAMETERS"."ALKALI/ACID_RECIRCULATION_TIME_PV",
                               DONE => "start dosing and recirculation_DB_1".DONE);
   END_IF;
   "IEC_Timer_0_DB_15".TP(IN := ("BUFFER"."MODE SELECTION" = 1) AND ("BUFFER".PROCESS = 140) AND "start dosing and recirculation_DB_1".DONE,
                          PT := T#1S);
   IF "IEC_Timer_0_DB_15".Q THEN "BUFFER".PROCESS := 150; END_IF;
   IF ("BUFFER".PROCESS = 150) OR ("BUFFER"."MODE SELECTION" = 0) THEN
       "start dosing and recirculation_DB_1".DONE := FALSE;
   END_IF;
   "start dosing and recirculation_DB_1".RESET := ("BUFFER".PROCESS = 150) OR ("BUFFER"."MODE SELECTION" = 0);
END_REGION

REGION Network 19: PH ACHIEVED OR NOT ACHIEVED BIT SET FOR POPUP.
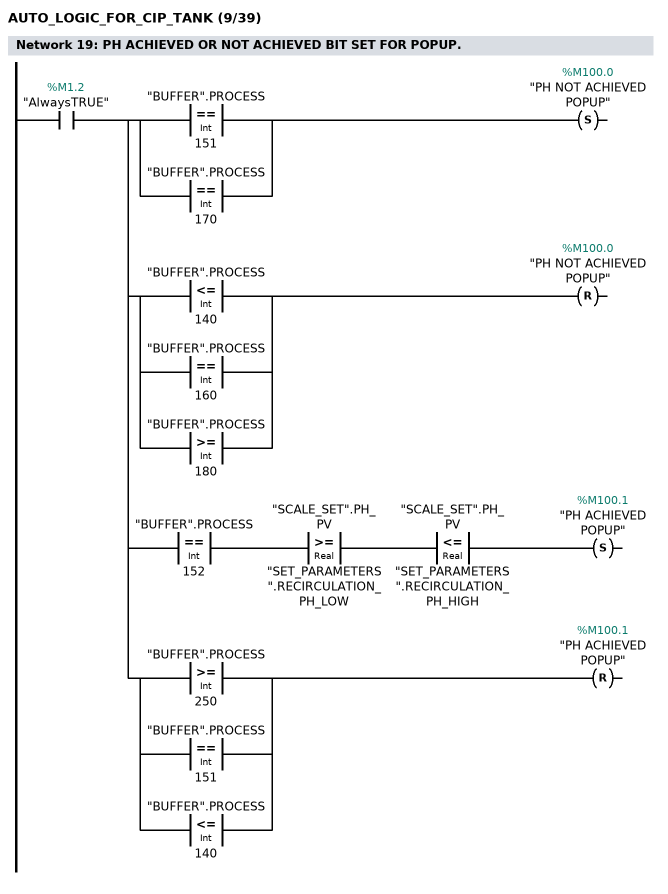
   RUNG wire#powerrail
      Contact( "AlwaysTRUE" )
      wire#w1
      { S7_Templates := "SrcType := Int" } EQ_Contact(in1 := "BUFFER".PROCESS, in2 := 151)
      wire#w2
      S_Coil( "PH NOT ACHIEVED POPUP" )
   END_RUNG
   RUNG wire#w1
      { S7_Templates := "SrcType := Int" } EQ_Contact(in1 := "BUFFER".PROCESS, in2 := 170)
   END_RUNG wire#w2
   RUNG wire#w1
      { S7_Templates := "SrcType := Int" } LE_Contact(in1 := "BUFFER".PROCESS, in2 := 140)
      wire#w3
      R_Coil( "PH NOT ACHIEVED POPUP" )
   END_RUNG
   RUNG wire#w1
      { S7_Templates := "SrcType := Int" } EQ_Contact(in1 := "BUFFER".PROCESS, in2 := 160)
   END_RUNG wire#w3
   RUNG wire#w1
      { S7_Templates := "SrcType := Int" } GE_Contact(in1 := "BUFFER".PROCESS, in2 := 180)
   END_RUNG wire#w3
   RUNG wire#w1
      { S7_Templates := "SrcType := Int" } EQ_Contact(in1 := "BUFFER".PROCESS, in2 := 152)
      { S7_Templates := "SrcType := Real" } GE_Contact(in1 := "SCALE_SET".PH_PV, in2 := "SET_PARAMETERS".RECIRCULATION_PH_LOW)
      { S7_Templates := "SrcType := Real" } LE_Contact(in1 := "SCALE_SET".PH_PV, in2 := "SET_PARAMETERS".RECIRCULATION_PH_HIGH)
      S_Coil( "PH ACHIEVED POPUP" )
   END_RUNG
   RUNG wire#w1
      { S7_Templates := "SrcType := Int" } GE_Contact(in1 := "BUFFER".PROCESS, in2 := 250)
      wire#w4
      R_Coil( "PH ACHIEVED POPUP" )
   END_RUNG
   RUNG wire#w1
      { S7_Templates := "SrcType := Int" } EQ_Contact(in1 := "BUFFER".PROCESS, in2 := 151)
   END_RUNG wire#w4
   RUNG wire#w1
      { S7_Templates := "SrcType := Int" } LE_Contact(in1 := "BUFFER".PROCESS, in2 := 140)
   END_RUNG wire#w4
   // the same network as SCL:
   IF "AlwaysTRUE" AND (("BUFFER".PROCESS = 151) OR ("BUFFER".PROCESS = 170)) THEN
       "PH NOT ACHIEVED POPUP" := TRUE;
   END_IF;
   IF "AlwaysTRUE" AND (("BUFFER".PROCESS <= 140) OR ("BUFFER".PROCESS = 160) OR ("BUFFER".PROCESS >= 180)) THEN
       "PH NOT ACHIEVED POPUP" := FALSE;
   END_IF;
   IF "AlwaysTRUE" AND ("BUFFER".PROCESS = 152) AND ("SCALE_SET".PH_PV >= "SET_PARAMETERS".RECIRCULATION_PH_LOW) AND ("SCALE_SET".PH_PV <= "SET_PARAMETERS".RECIRCULATION_PH_HIGH) THEN
       "PH ACHIEVED POPUP" := TRUE;
   END_IF;
   IF "AlwaysTRUE" AND (("BUFFER".PROCESS >= 250) OR ("BUFFER".PROCESS = 151) OR ("BUFFER".PROCESS <= 140)) THEN
       "PH ACHIEVED POPUP" := FALSE;
   END_IF;
END_REGION

REGION Network 20: ALKALI/ACID_PH CHECKING_TIME_
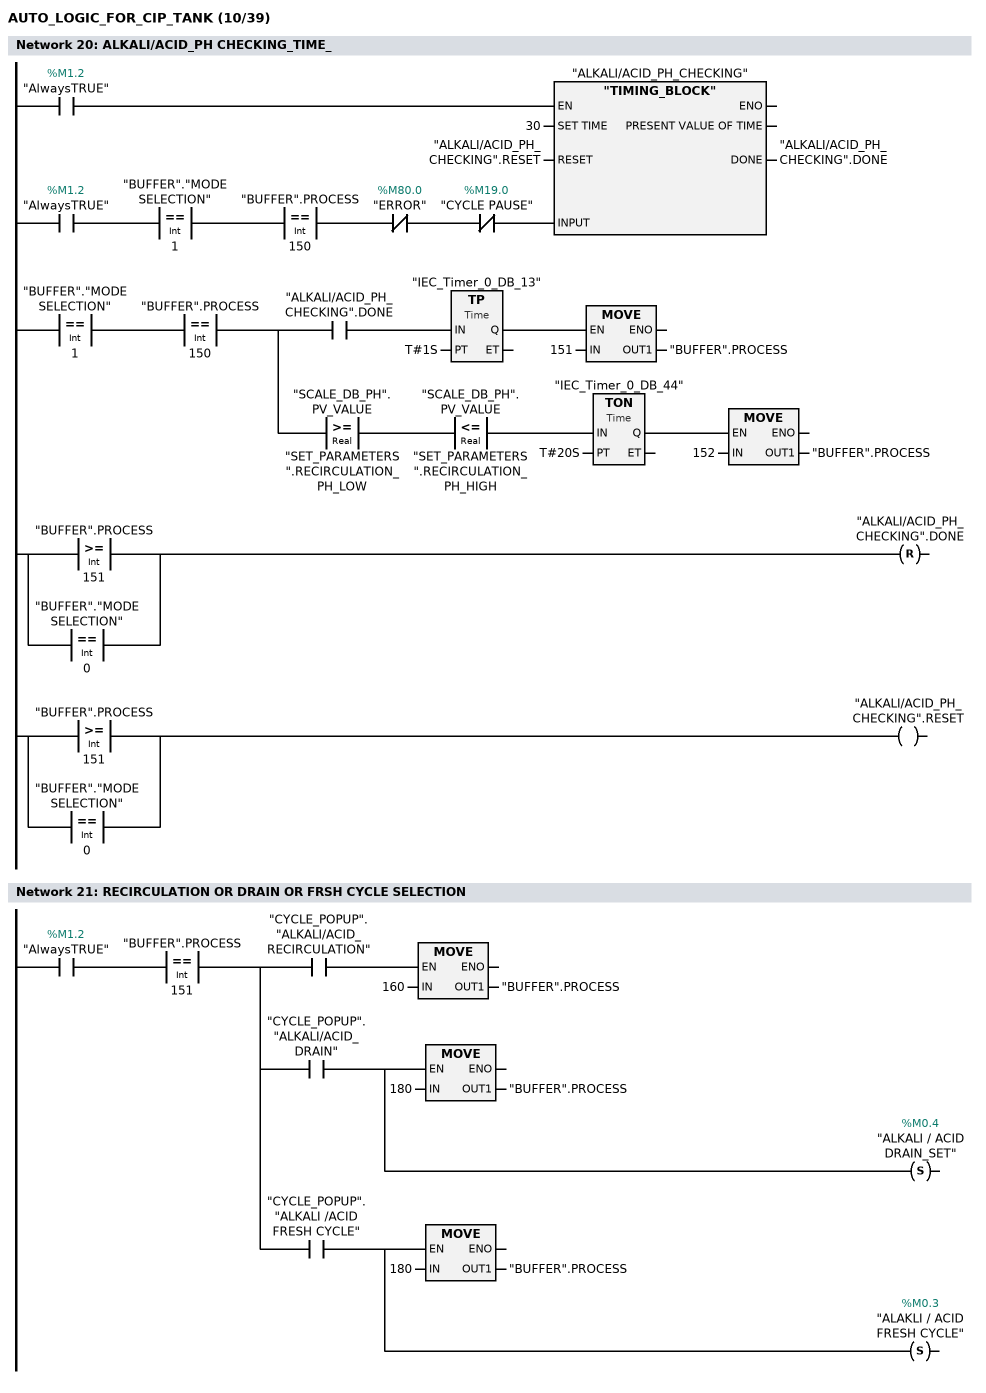
   RUNG wire#powerrail
      Contact( "AlwaysTRUE" )
      "ALKALI/ACID_PH_CHECKING"(INPUT := wire#w1, "SET TIME" := 30, RESET := "ALKALI/ACID_PH_CHECKING".RESET, "PRESENT VALUE OF TIME" =>, DONE => "ALKALI/ACID_PH_CHECKING".DONE)
   END_RUNG
   RUNG wire#powerrail
      Contact( "AlwaysTRUE" )
      { S7_Templates := "SrcType := Int" } EQ_Contact(in1 := "BUFFER"."MODE SELECTION", in2 := 1)
      { S7_Templates := "SrcType := Int" } EQ_Contact(in1 := "BUFFER".PROCESS, in2 := 150)
      I_Contact( "ERROR" )
      I_Contact( "CYCLE PAUSE" )
   END_RUNG wire#w1
   RUNG wire#powerrail
      { S7_Templates := "SrcType := Int" } EQ_Contact(in1 := "BUFFER"."MODE SELECTION", in2 := 1)
      { S7_Templates := "SrcType := Int" } EQ_Contact(in1 := "BUFFER".PROCESS, in2 := 150)
      wire#w2
      Contact( "ALKALI/ACID_PH_CHECKING".DONE )
      { S7_Templates := "time_type := Time" } "IEC_Timer_0_DB_13".TP(pt := T#1S, et =>)
      Move(in := 151, out1 => "BUFFER".PROCESS)
   END_RUNG
   RUNG wire#w2
      { S7_Templates := "SrcType := Real" } GE_Contact(in1 := "SCALE_DB_PH".PV_VALUE, in2 := "SET_PARAMETERS".RECIRCULATION_PH_LOW)
      { S7_Templates := "SrcType := Real" } LE_Contact(in1 := "SCALE_DB_PH".PV_VALUE, in2 := "SET_PARAMETERS".RECIRCULATION_PH_HIGH)
      { S7_Templates := "time_type := Time" } "IEC_Timer_0_DB_44".TON(pt := T#20S, et =>)
      Move(in := 152, out1 => "BUFFER".PROCESS)
   END_RUNG
   RUNG wire#powerrail
      { S7_Templates := "SrcType := Int" } GE_Contact(in1 := "BUFFER".PROCESS, in2 := 151)
      wire#w3
      R_Coil( "ALKALI/ACID_PH_CHECKING".DONE )
   END_RUNG
   RUNG wire#powerrail
      { S7_Templates := "SrcType := Int" } EQ_Contact(in1 := "BUFFER"."MODE SELECTION", in2 := 0)
   END_RUNG wire#w3
   RUNG wire#powerrail
      { S7_Templates := "SrcType := Int" } GE_Contact(in1 := "BUFFER".PROCESS, in2 := 151)
      wire#w4
      Coil( "ALKALI/ACID_PH_CHECKING".RESET )
   END_RUNG
   RUNG wire#powerrail
      { S7_Templates := "SrcType := Int" } EQ_Contact(in1 := "BUFFER"."MODE SELECTION", in2 := 0)
   END_RUNG wire#w4
   // the same network as SCL:
   IF "AlwaysTRUE" THEN
       "ALKALI/ACID_PH_CHECKING"("SET TIME" := 30,   // "TIMING_BLOCK"
                               RESET := "ALKALI/ACID_PH_CHECKING".RESET,
                               INPUT := "AlwaysTRUE" AND ("BUFFER"."MODE SELECTION" = 1) AND ("BUFFER".PROCESS = 150) AND NOT "ERROR" AND NOT "CYCLE PAUSE",
                               DONE => "ALKALI/ACID_PH_CHECKING".DONE);
   END_IF;
   #_w1 := ("BUFFER"."MODE SELECTION" = 1) AND ("BUFFER".PROCESS = 150);
   "IEC_Timer_0_DB_13".TP(IN := #_w1 AND "ALKALI/ACID_PH_CHECKING".DONE, PT := T#1S);
   IF "IEC_Timer_0_DB_13".Q THEN "BUFFER".PROCESS := 151; END_IF;
   "IEC_Timer_0_DB_44".TON(IN := #_w1 AND ("SCALE_DB_PH".PV_VALUE >= "SET_PARAMETERS".RECIRCULATION_PH_LOW) AND ("SCALE_DB_PH".PV_VALUE <= "SET_PARAMETERS".RECIRCULATION_PH_HIGH),
                           PT := T#20S);
   IF "IEC_Timer_0_DB_44".Q THEN "BUFFER".PROCESS := 152; END_IF;
   IF ("BUFFER".PROCESS >= 151) OR ("BUFFER"."MODE SELECTION" = 0) THEN
       "ALKALI/ACID_PH_CHECKING".DONE := FALSE;
   END_IF;
   "ALKALI/ACID_PH_CHECKING".RESET := ("BUFFER".PROCESS >= 151) OR ("BUFFER"."MODE SELECTION" = 0);
END_REGION

REGION Network 21: RECIRCULATION OR DRAIN OR FRSH CYCLE SELECTION
   RUNG wire#powerrail
      Contact( "AlwaysTRUE" )
      { S7_Templates := "SrcType := Int" } EQ_Contact(in1 := "BUFFER".PROCESS, in2 := 151)
      wire#w1
      Contact( "CYCLE_POPUP"."ALKALI/ACID_RECIRCULATION" )
      Move(in := 160, out1 => "BUFFER".PROCESS)
   END_RUNG
   RUNG wire#w1
      Contact( "CYCLE_POPUP"."ALKALI/ACID_DRAIN" )
      wire#w2
      Move(in := 180, out1 => "BUFFER".PROCESS)
   END_RUNG
   RUNG wire#w2
      S_Coil( "ALKALI / ACID DRAIN_SET" )
   END_RUNG
   RUNG wire#w1
      Contact( "CYCLE_POPUP"."ALKALI /ACID FRESH CYCLE" )
      wire#w3
      Move(in := 180, out1 => "BUFFER".PROCESS)
   END_RUNG
   RUNG wire#w3
      S_Coil( "ALAKLI / ACID FRESH CYCLE" )
   END_RUNG
   // the same network as SCL:
   #_w1 := "AlwaysTRUE" AND ("BUFFER".PROCESS = 151);
   IF #_w1 AND "CYCLE_POPUP"."ALKALI/ACID_RECIRCULATION" THEN "BUFFER".PROCESS := 160; END_IF;
   IF #_w1 AND "CYCLE_POPUP"."ALKALI/ACID_DRAIN" THEN
       "BUFFER".PROCESS := 180;
       "ALKALI / ACID DRAIN_SET" := TRUE;
   END_IF;
   IF #_w1 AND "CYCLE_POPUP"."ALKALI /ACID FRESH CYCLE" THEN
       "BUFFER".PROCESS := 180;
       "ALAKLI / ACID FRESH CYCLE" := TRUE;
   END_IF;
END_REGION

REGION Network 22: PH ACHIEVED GONG TO DRAIN
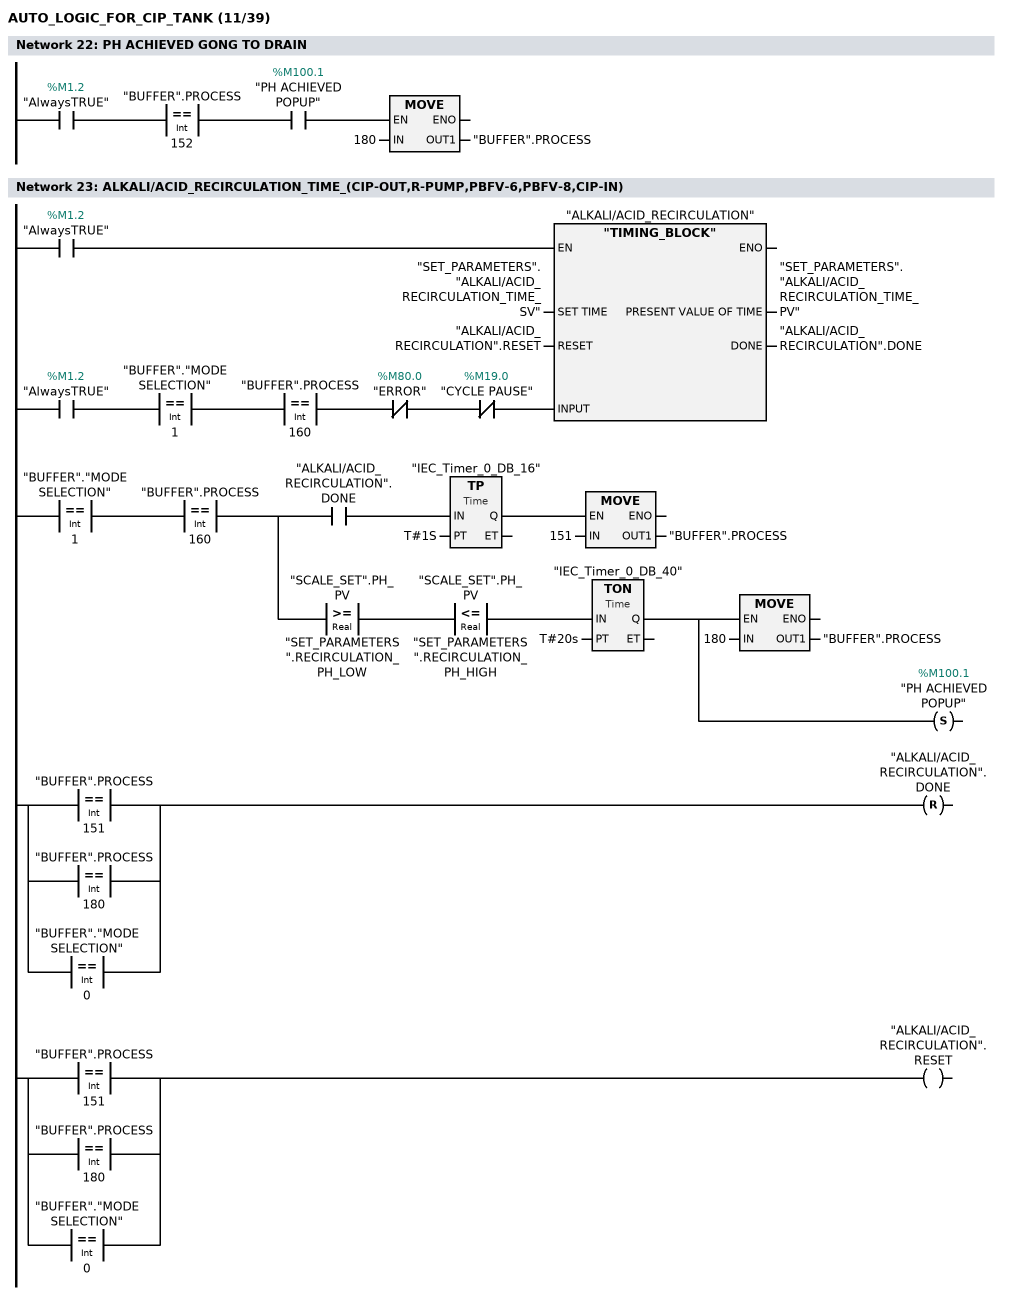
   RUNG wire#powerrail
      Contact( "AlwaysTRUE" )
      { S7_Templates := "SrcType := Int" } EQ_Contact(in1 := "BUFFER".PROCESS, in2 := 152)
      Contact( "PH ACHIEVED POPUP" )
      Move(in := 180, out1 => "BUFFER".PROCESS)
   END_RUNG
   // the same network as SCL:
   IF "AlwaysTRUE" AND ("BUFFER".PROCESS = 152) AND "PH ACHIEVED POPUP" THEN "BUFFER".PROCESS := 180; END_IF;
END_REGION

REGION Network 23: ALKALI/ACID_RECIRCULATION_TIME_(CIP-OUT,R-PUMP,PBFV-6,PBFV-8,CIP-IN)
   RUNG wire#powerrail
      Contact( "AlwaysTRUE" )
      "ALKALI/ACID_RECIRCULATION"(INPUT := wire#w1, "SET TIME" := "SET_PARAMETERS"."ALKALI/ACID_RECIRCULATION_TIME_SV", RESET := "ALKALI/ACID_RECIRCULATION".RESET, "PRESENT VALUE OF TIME" => "SET_PARAMETERS"."ALKALI/ACID_RECIRCULATION_TIME_PV", DONE => "ALKALI/ACID_RECIRCULATION".DONE)
   END_RUNG
   RUNG wire#powerrail
      Contact( "AlwaysTRUE" )
      { S7_Templates := "SrcType := Int" } EQ_Contact(in1 := "BUFFER"."MODE SELECTION", in2 := 1)
      { S7_Templates := "SrcType := Int" } EQ_Contact(in1 := "BUFFER".PROCESS, in2 := 160)
      I_Contact( "ERROR" )
      I_Contact( "CYCLE PAUSE" )
   END_RUNG wire#w1
   RUNG wire#powerrail
      { S7_Templates := "SrcType := Int" } EQ_Contact(in1 := "BUFFER"."MODE SELECTION", in2 := 1)
      { S7_Templates := "SrcType := Int" } EQ_Contact(in1 := "BUFFER".PROCESS, in2 := 160)
      wire#w2
      Contact( "ALKALI/ACID_RECIRCULATION".DONE )
      { S7_Templates := "time_type := Time" } "IEC_Timer_0_DB_16".TP(pt := T#1S, et =>)
      Move(in := 151, out1 => "BUFFER".PROCESS)
   END_RUNG
   RUNG wire#w2
      { S7_Templates := "SrcType := Real" } GE_Contact(in1 := "SCALE_SET".PH_PV, in2 := "SET_PARAMETERS".RECIRCULATION_PH_LOW)
      { S7_Templates := "SrcType := Real" } LE_Contact(in1 := "SCALE_SET".PH_PV, in2 := "SET_PARAMETERS".RECIRCULATION_PH_HIGH)
      { S7_Templates := "time_type := Time" } "IEC_Timer_0_DB_40".TON(pt := T#20s, et =>)
      wire#w3
      Move(in := 180, out1 => "BUFFER".PROCESS)
   END_RUNG
   RUNG wire#w3
      S_Coil( "PH ACHIEVED POPUP" )
   END_RUNG
   RUNG wire#powerrail
      { S7_Templates := "SrcType := Int" } EQ_Contact(in1 := "BUFFER".PROCESS, in2 := 151)
      wire#w4
      R_Coil( "ALKALI/ACID_RECIRCULATION".DONE )
   END_RUNG
   RUNG wire#powerrail
      { S7_Templates := "SrcType := Int" } EQ_Contact(in1 := "BUFFER".PROCESS, in2 := 180)
   END_RUNG wire#w4
   RUNG wire#powerrail
      { S7_Templates := "SrcType := Int" } EQ_Contact(in1 := "BUFFER"."MODE SELECTION", in2 := 0)
   END_RUNG wire#w4
   RUNG wire#powerrail
      { S7_Templates := "SrcType := Int" } EQ_Contact(in1 := "BUFFER".PROCESS, in2 := 151)
      wire#w5
      Coil( "ALKALI/ACID_RECIRCULATION".RESET )
   END_RUNG
   RUNG wire#powerrail
      { S7_Templates := "SrcType := Int" } EQ_Contact(in1 := "BUFFER".PROCESS, in2 := 180)
   END_RUNG wire#w5
   RUNG wire#powerrail
      { S7_Templates := "SrcType := Int" } EQ_Contact(in1 := "BUFFER"."MODE SELECTION", in2 := 0)
   END_RUNG wire#w5
   // the same network as SCL:
   IF "AlwaysTRUE" THEN
       "ALKALI/ACID_RECIRCULATION"("SET TIME" := "SET_PARAMETERS"."ALKALI/ACID_RECIRCULATION_TIME_SV",   // "TIMING_BLOCK"
                               RESET := "ALKALI/ACID_RECIRCULATION".RESET,
                               INPUT := "AlwaysTRUE" AND ("BUFFER"."MODE SELECTION" = 1) AND ("BUFFER".PROCESS = 160) AND NOT "ERROR" AND NOT "CYCLE PAUSE",
                               "PRESENT VALUE OF TIME" => "SET_PARAMETERS"."ALKALI/ACID_RECIRCULATION_TIME_PV",
                               DONE => "ALKALI/ACID_RECIRCULATION".DONE);
   END_IF;
   #_w1 := ("BUFFER"."MODE SELECTION" = 1) AND ("BUFFER".PROCESS = 160);
   "IEC_Timer_0_DB_16".TP(IN := #_w1 AND "ALKALI/ACID_RECIRCULATION".DONE, PT := T#1S);
   IF "IEC_Timer_0_DB_16".Q THEN "BUFFER".PROCESS := 151; END_IF;
   "IEC_Timer_0_DB_40".TON(IN := #_w1 AND ("SCALE_SET".PH_PV >= "SET_PARAMETERS".RECIRCULATION_PH_LOW) AND ("SCALE_SET".PH_PV <= "SET_PARAMETERS".RECIRCULATION_PH_HIGH),
                           PT := T#20s);
   IF "IEC_Timer_0_DB_40".Q THEN
       "BUFFER".PROCESS := 180;
       "PH ACHIEVED POPUP" := TRUE;
   END_IF;
   IF ("BUFFER".PROCESS = 151) OR ("BUFFER".PROCESS = 180) OR ("BUFFER"."MODE SELECTION" = 0) THEN
       "ALKALI/ACID_RECIRCULATION".DONE := FALSE;
   END_IF;
   "ALKALI/ACID_RECIRCULATION".RESET := ("BUFFER".PROCESS = 151) OR ("BUFFER".PROCESS = 180) OR ("BUFFER"."MODE SELECTION" = 0);
END_REGION

REGION Network 24: ALKALI/ACID_DRAIN_TIME_(CIP-OUT,R_PUMP,PBFV-11)
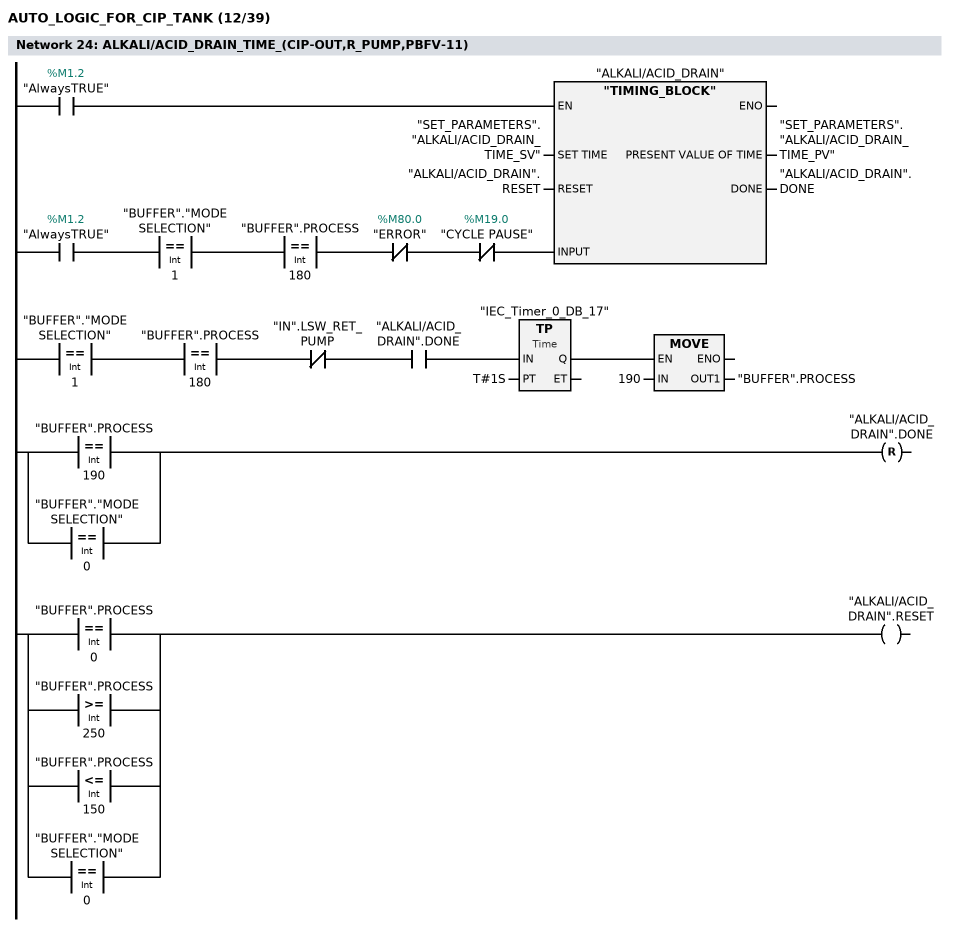
   RUNG wire#powerrail
      Contact( "AlwaysTRUE" )
      "ALKALI/ACID_DRAIN"(INPUT := wire#w1, "SET TIME" := "SET_PARAMETERS"."ALKALI/ACID_DRAIN_TIME_SV", RESET := "ALKALI/ACID_DRAIN".RESET, "PRESENT VALUE OF TIME" => "SET_PARAMETERS"."ALKALI/ACID_DRAIN_TIME_PV", DONE => "ALKALI/ACID_DRAIN".DONE)
   END_RUNG
   RUNG wire#powerrail
      Contact( "AlwaysTRUE" )
      { S7_Templates := "SrcType := Int" } EQ_Contact(in1 := "BUFFER"."MODE SELECTION", in2 := 1)
      { S7_Templates := "SrcType := Int" } EQ_Contact(in1 := "BUFFER".PROCESS, in2 := 180)
      I_Contact( "ERROR" )
      I_Contact( "CYCLE PAUSE" )
   END_RUNG wire#w1
   RUNG wire#powerrail
      { S7_Templates := "SrcType := Int" } EQ_Contact(in1 := "BUFFER"."MODE SELECTION", in2 := 1)
      { S7_Templates := "SrcType := Int" } EQ_Contact(in1 := "BUFFER".PROCESS, in2 := 180)
      I_Contact( "IN".LSW_RET_PUMP )
      Contact( "ALKALI/ACID_DRAIN".DONE )
      { S7_Templates := "time_type := Time" } "IEC_Timer_0_DB_17".TP(pt := T#1S, et =>)
      Move(in := 190, out1 => "BUFFER".PROCESS)
   END_RUNG
   RUNG wire#powerrail
      { S7_Templates := "SrcType := Int" } EQ_Contact(in1 := "BUFFER".PROCESS, in2 := 190)
      wire#w2
      R_Coil( "ALKALI/ACID_DRAIN".DONE )
   END_RUNG
   RUNG wire#powerrail
      { S7_Templates := "SrcType := Int" } EQ_Contact(in1 := "BUFFER"."MODE SELECTION", in2 := 0)
   END_RUNG wire#w2
   RUNG wire#powerrail
      { S7_Templates := "SrcType := Int" } EQ_Contact(in1 := "BUFFER".PROCESS, in2 := 0)
      wire#w3
      Coil( "ALKALI/ACID_DRAIN".RESET )
   END_RUNG
   RUNG wire#powerrail
      { S7_Templates := "SrcType := Int" } GE_Contact(in1 := "BUFFER".PROCESS, in2 := 250)
   END_RUNG wire#w3
   RUNG wire#powerrail
      { S7_Templates := "SrcType := Int" } LE_Contact(in1 := "BUFFER".PROCESS, in2 := 150)
   END_RUNG wire#w3
   RUNG wire#powerrail
      { S7_Templates := "SrcType := Int" } EQ_Contact(in1 := "BUFFER"."MODE SELECTION", in2 := 0)
   END_RUNG wire#w3
   // the same network as SCL:
   IF "AlwaysTRUE" THEN
       "ALKALI/ACID_DRAIN"("SET TIME" := "SET_PARAMETERS"."ALKALI/ACID_DRAIN_TIME_SV",   // "TIMING_BLOCK"
                           RESET := "ALKALI/ACID_DRAIN".RESET,
                           INPUT := "AlwaysTRUE" AND ("BUFFER"."MODE SELECTION" = 1) AND ("BUFFER".PROCESS = 180) AND NOT "ERROR" AND NOT "CYCLE PAUSE",
                           "PRESENT VALUE OF TIME" => "SET_PARAMETERS"."ALKALI/ACID_DRAIN_TIME_PV",
                           DONE => "ALKALI/ACID_DRAIN".DONE);
   END_IF;
   "IEC_Timer_0_DB_17".TP(IN := ("BUFFER"."MODE SELECTION" = 1) AND ("BUFFER".PROCESS = 180) AND NOT "IN".LSW_RET_PUMP AND "ALKALI/ACID_DRAIN".DONE,
                          PT := T#1S);
   IF "IEC_Timer_0_DB_17".Q THEN "BUFFER".PROCESS := 190; END_IF;
   IF ("BUFFER".PROCESS = 190) OR ("BUFFER"."MODE SELECTION" = 0) THEN
       "ALKALI/ACID_DRAIN".DONE := FALSE;
   END_IF;
   "ALKALI/ACID_DRAIN".RESET := ("BUFFER".PROCESS = 0) OR ("BUFFER".PROCESS >= 250) OR ("BUFFER".PROCESS <= 150) OR ("BUFFER"."MODE SELECTION" = 0);
END_REGION

REGION Network 25: ALKALI/ACID_PUMP_CHASING_TIME_(PBFV-12,PBFV13)
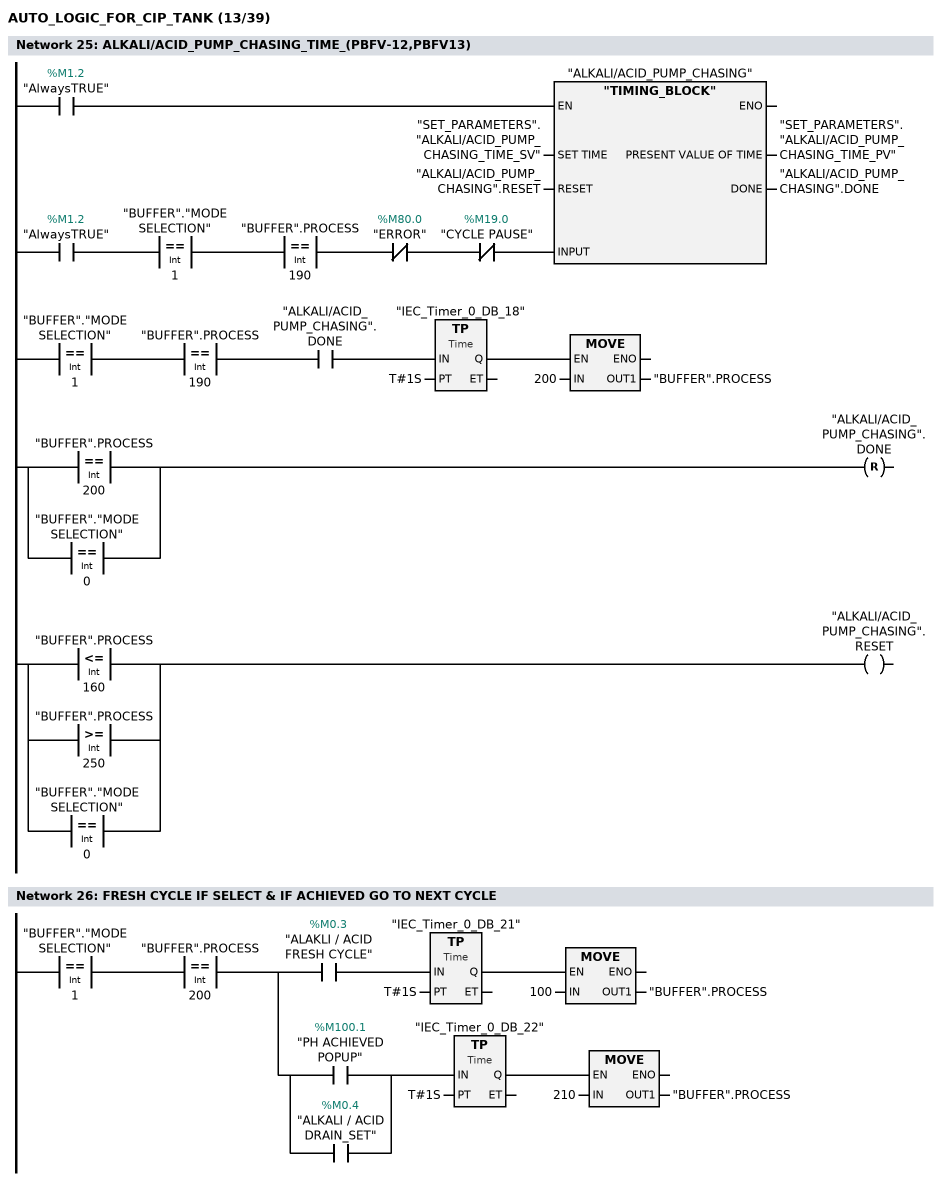
   RUNG wire#powerrail
      Contact( "AlwaysTRUE" )
      "ALKALI/ACID_PUMP_CHASING"(INPUT := wire#w1, "SET TIME" := "SET_PARAMETERS"."ALKALI/ACID_PUMP_CHASING_TIME_SV", RESET := "ALKALI/ACID_PUMP_CHASING".RESET, "PRESENT VALUE OF TIME" => "SET_PARAMETERS"."ALKALI/ACID_PUMP_CHASING_TIME_PV", DONE => "ALKALI/ACID_PUMP_CHASING".DONE)
   END_RUNG
   RUNG wire#powerrail
      Contact( "AlwaysTRUE" )
      { S7_Templates := "SrcType := Int" } EQ_Contact(in1 := "BUFFER"."MODE SELECTION", in2 := 1)
      { S7_Templates := "SrcType := Int" } EQ_Contact(in1 := "BUFFER".PROCESS, in2 := 190)
      I_Contact( "ERROR" )
      I_Contact( "CYCLE PAUSE" )
   END_RUNG wire#w1
   RUNG wire#powerrail
      { S7_Templates := "SrcType := Int" } EQ_Contact(in1 := "BUFFER"."MODE SELECTION", in2 := 1)
      { S7_Templates := "SrcType := Int" } EQ_Contact(in1 := "BUFFER".PROCESS, in2 := 190)
      Contact( "ALKALI/ACID_PUMP_CHASING".DONE )
      { S7_Templates := "time_type := Time" } "IEC_Timer_0_DB_18".TP(pt := T#1S, et =>)
      Move(in := 200, out1 => "BUFFER".PROCESS)
   END_RUNG
   RUNG wire#powerrail
      { S7_Templates := "SrcType := Int" } EQ_Contact(in1 := "BUFFER".PROCESS, in2 := 200)
      wire#w2
      R_Coil( "ALKALI/ACID_PUMP_CHASING".DONE )
   END_RUNG
   RUNG wire#powerrail
      { S7_Templates := "SrcType := Int" } EQ_Contact(in1 := "BUFFER"."MODE SELECTION", in2 := 0)
   END_RUNG wire#w2
   RUNG wire#powerrail
      { S7_Templates := "SrcType := Int" } LE_Contact(in1 := "BUFFER".PROCESS, in2 := 160)
      wire#w3
      Coil( "ALKALI/ACID_PUMP_CHASING".RESET )
   END_RUNG
   RUNG wire#powerrail
      { S7_Templates := "SrcType := Int" } GE_Contact(in1 := "BUFFER".PROCESS, in2 := 250)
   END_RUNG wire#w3
   RUNG wire#powerrail
      { S7_Templates := "SrcType := Int" } EQ_Contact(in1 := "BUFFER"."MODE SELECTION", in2 := 0)
   END_RUNG wire#w3
   // the same network as SCL:
   IF "AlwaysTRUE" THEN
       "ALKALI/ACID_PUMP_CHASING"("SET TIME" := "SET_PARAMETERS"."ALKALI/ACID_PUMP_CHASING_TIME_SV",   // "TIMING_BLOCK"
                               RESET := "ALKALI/ACID_PUMP_CHASING".RESET,
                               INPUT := "AlwaysTRUE" AND ("BUFFER"."MODE SELECTION" = 1) AND ("BUFFER".PROCESS = 190) AND NOT "ERROR" AND NOT "CYCLE PAUSE",
                               "PRESENT VALUE OF TIME" => "SET_PARAMETERS"."ALKALI/ACID_PUMP_CHASING_TIME_PV",
                               DONE => "ALKALI/ACID_PUMP_CHASING".DONE);
   END_IF;
   "IEC_Timer_0_DB_18".TP(IN := ("BUFFER"."MODE SELECTION" = 1) AND ("BUFFER".PROCESS = 190) AND "ALKALI/ACID_PUMP_CHASING".DONE,
                          PT := T#1S);
   IF "IEC_Timer_0_DB_18".Q THEN "BUFFER".PROCESS := 200; END_IF;
   IF ("BUFFER".PROCESS = 200) OR ("BUFFER"."MODE SELECTION" = 0) THEN
       "ALKALI/ACID_PUMP_CHASING".DONE := FALSE;
   END_IF;
   "ALKALI/ACID_PUMP_CHASING".RESET := ("BUFFER".PROCESS <= 160) OR ("BUFFER".PROCESS >= 250) OR ("BUFFER"."MODE SELECTION" = 0);
END_REGION

REGION Network 26: FRESH CYCLE IF SELECT & IF ACHIEVED GO TO NEXT CYCLE
   RUNG wire#powerrail
      { S7_Templates := "SrcType := Int" } EQ_Contact(in1 := "BUFFER"."MODE SELECTION", in2 := 1)
      { S7_Templates := "SrcType := Int" } EQ_Contact(in1 := "BUFFER".PROCESS, in2 := 200)
      wire#w1
      Contact( "ALAKLI / ACID FRESH CYCLE" )
      { S7_Templates := "time_type := Time" } "IEC_Timer_0_DB_21".TP(pt := T#1S, et =>)
      Move(in := 100, out1 => "BUFFER".PROCESS)
   END_RUNG
   RUNG wire#w1
      Contact( "PH ACHIEVED POPUP" )
      wire#w2
      { S7_Templates := "time_type := Time" } "IEC_Timer_0_DB_22".TP(pt := T#1S, et =>)
      Move(in := 210, out1 => "BUFFER".PROCESS)
   END_RUNG
   RUNG wire#w1
      Contact( "ALKALI / ACID DRAIN_SET" )
   END_RUNG wire#w2
   // the same network as SCL:
   #_w1 := ("BUFFER"."MODE SELECTION" = 1) AND ("BUFFER".PROCESS = 200);
   "IEC_Timer_0_DB_21".TP(IN := #_w1 AND "ALAKLI / ACID FRESH CYCLE", PT := T#1S);
   IF "IEC_Timer_0_DB_21".Q THEN "BUFFER".PROCESS := 100; END_IF;
   "IEC_Timer_0_DB_22".TP(IN := #_w1 AND ("PH ACHIEVED POPUP" OR "ALKALI / ACID DRAIN_SET"), PT := T#1S);
   IF "IEC_Timer_0_DB_22".Q THEN "BUFFER".PROCESS := 210; END_IF;
END_REGION

REGION Network 30: NEXT_CYCLE(RINSE-2) POPUP
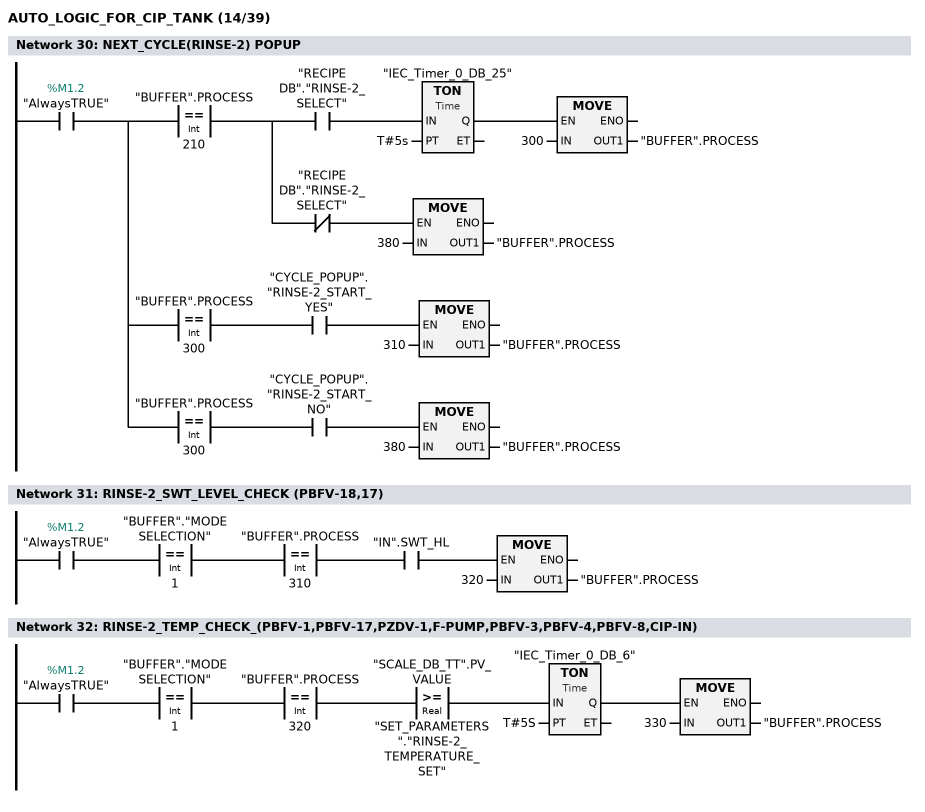
   RUNG wire#powerrail
      Contact( "AlwaysTRUE" )
      wire#w1
      { S7_Templates := "SrcType := Int" } EQ_Contact(in1 := "BUFFER".PROCESS, in2 := 210)
      wire#w2
      Contact( "RECIPE DB"."RINSE-2_SELECT" )
      { S7_Templates := "time_type := Time" } "IEC_Timer_0_DB_25".TON(pt := T#5s, et =>)
      Move(in := 300, out1 => "BUFFER".PROCESS)
   END_RUNG
   RUNG wire#w2
      I_Contact( "RECIPE DB"."RINSE-2_SELECT" )
      Move(in := 380, out1 => "BUFFER".PROCESS)
   END_RUNG
   RUNG wire#w1
      { S7_Templates := "SrcType := Int" } EQ_Contact(in1 := "BUFFER".PROCESS, in2 := 300)
      Contact( "CYCLE_POPUP"."RINSE-2_START_YES" )
      Move(in := 310, out1 => "BUFFER".PROCESS)
   END_RUNG
   RUNG wire#w1
      { S7_Templates := "SrcType := Int" } EQ_Contact(in1 := "BUFFER".PROCESS, in2 := 300)
      Contact( "CYCLE_POPUP"."RINSE-2_START_NO" )
      Move(in := 380, out1 => "BUFFER".PROCESS)
   END_RUNG
   // the same network as SCL:
   #_w1 := "AlwaysTRUE" AND ("BUFFER".PROCESS = 210);
   "IEC_Timer_0_DB_25".TON(IN := #_w1 AND "RECIPE DB"."RINSE-2_SELECT", PT := T#5s);
   IF "IEC_Timer_0_DB_25".Q THEN "BUFFER".PROCESS := 300; END_IF;
   IF #_w1 AND NOT "RECIPE DB"."RINSE-2_SELECT" THEN "BUFFER".PROCESS := 380; END_IF;
   IF "AlwaysTRUE" AND ("BUFFER".PROCESS = 300) AND "CYCLE_POPUP"."RINSE-2_START_YES" THEN
       "BUFFER".PROCESS := 310;
   END_IF;
   IF "AlwaysTRUE" AND ("BUFFER".PROCESS = 300) AND "CYCLE_POPUP"."RINSE-2_START_NO" THEN
       "BUFFER".PROCESS := 380;
   END_IF;
END_REGION

REGION Network 31: RINSE-2_SWT_LEVEL_CHECK (PBFV-18,17)
   RUNG wire#powerrail
      Contact( "AlwaysTRUE" )
      { S7_Templates := "SrcType := Int" } EQ_Contact(in1 := "BUFFER"."MODE SELECTION", in2 := 1)
      { S7_Templates := "SrcType := Int" } EQ_Contact(in1 := "BUFFER".PROCESS, in2 := 310)
      Contact( "IN".SWT_HL )
      Move(in := 320, out1 => "BUFFER".PROCESS)
   END_RUNG
   // the same network as SCL:
   IF "AlwaysTRUE" AND ("BUFFER"."MODE SELECTION" = 1) AND ("BUFFER".PROCESS = 310) AND "IN".SWT_HL THEN
       "BUFFER".PROCESS := 320;
   END_IF;
END_REGION

REGION Network 32: RINSE-2_TEMP_CHECK_(PBFV-1,PBFV-17,PZDV-1,F-PUMP,PBFV-3,PBFV-4,PBFV-8,CIP-IN)
   RUNG wire#powerrail
      Contact( "AlwaysTRUE" )
      { S7_Templates := "SrcType := Int" } EQ_Contact(in1 := "BUFFER"."MODE SELECTION", in2 := 1)
      { S7_Templates := "SrcType := Int" } EQ_Contact(in1 := "BUFFER".PROCESS, in2 := 320)
      { S7_Templates := "SrcType := Real" } GE_Contact(in1 := "SCALE_DB_TT".PV_VALUE, in2 := "SET_PARAMETERS"."RINSE-2_TEMPERATURE_SET")
      { S7_Templates := "time_type := Time" } "IEC_Timer_0_DB_6".TON(pt := T#5S, et =>)
      Move(in := 330, out1 => "BUFFER".PROCESS)
   END_RUNG
   // the same network as SCL:
   "IEC_Timer_0_DB_6".TON(IN := "AlwaysTRUE" AND ("BUFFER"."MODE SELECTION" = 1) AND ("BUFFER".PROCESS = 320) AND ("SCALE_DB_TT".PV_VALUE >= "SET_PARAMETERS"."RINSE-2_TEMPERATURE_SET"),
                          PT := T#5S);
   IF "IEC_Timer_0_DB_6".Q THEN "BUFFER".PROCESS := 330; END_IF;
END_REGION

